SPLINE
SPL {X  -158.454, Y  +360.384, Z    +0.000, E1  +340.634, E3 -446476.060}
SPL {X  -159.737, Y  +373.507, Z    +0.000, E1  +349.689, E3 -446498.095}
SPL {X  -159.990, Y  +382.574, Z    +0.000, E1  +355.537, E3 -446504.783}
SPL {X  -159.990, Y  +389.909, Z    +0.000, E1  +360.662, E3 -446508.797}
SPL {X  -159.990, Y  +396.289, Z    +0.000, E1  +365.500, E3 -446512.577}
SPL {X  -159.990, Y  +407.941, Z    +0.000, E1  +374.126, E3 -446523.914}
SPL {X  -159.990, Y  +418.671, Z    +0.000, E1  +379.855, E3 -446543.330}
SPL {X  -159.990, Y  +429.878, Z    +0.000, E1  +383.330, E3 -446573.386}
SPL {X  -159.990, Y  +432.103, Z    +0.000, E1  +383.301, E3 -446584.404}
SPL {X  -159.990, Y  +434.188, Z    +0.000, E1  +383.325, E3 -446594.601}
SPL {X  -159.990, Y  +437.007, Z    +0.000, E1  +383.323, E3 -446608.492}
SPL {X  -159.990, Y  +439.778, Z    +0.000, E1  +383.323, E3 -446622.124}
SPL {X  -159.990, Y  +442.010, Z    +0.000, E1  +383.308, E3 -446633.145}
SPL {X  -159.990, Y  +443.729, Z    +0.000, E1  +383.310, E3 -446641.601}
SPL {X  -159.990, Y  +446.037, Z    +0.000, E1  +383.324, E3 -446652.938}
SPL {X  -159.990, Y  +448.341, Z    +0.000, E1  +383.317, E3 -446664.256}
SPL {X  -159.990, Y  +450.345, Z    +0.000, E1  +383.316, E3 -446674.134}
SPL {X  -159.990, Y  +452.828, Z    +0.000, E1  +383.330, E3 -446686.333}
SPL {X  -159.990, Y  +456.338, Z    +0.000, E1  +383.359, E3 -446703.525}
SPL {X  -159.990, Y  +459.480, Z    +0.000, E1  +383.323, E3 -446719.067}
SPL {X  -159.990, Y  +461.803, Z    +0.000, E1  +383.322, E3 -446730.502}
SPL {X  -159.990, Y  +464.971, Z    +0.000, E1  +383.357, E3 -446746.008}
SPL {X  -159.990, Y  +467.934, Z    +0.000, E1  +383.321, E3 -446760.665}
SPL {X  -159.990, Y  +469.939, Z    +0.000, E1  +383.319, E3 -446770.527}
SPL {X  -159.990, Y  +472.144, Z    +0.000, E1  +383.327, E3 -446781.378}
SPL {X  -159.990, Y  +474.152, Z    +0.000, E1  +383.309, E3 -446791.330}
SPL {X  -159.990, Y  +476.560, Z    +0.000, E1  +383.332, E3 -446803.138}
SPL {X  -159.990, Y  +478.770, Z    +0.000, E1  +383.306, E3 -446814.063}
SPL {X  -159.990, Y  +480.905, Z    +0.000, E1  +383.327, E3 -446824.531}
SPL {X  -159.990, Y  +484.251, Z    +0.000, E1  +383.352, E3 -446840.947}
SPL {X  -159.990, Y  +488.031, Z    +0.000, E1  +383.345, E3 -446859.579}
SPL {X  -159.990, Y  +491.121, Z    +0.000, E1  +383.323, E3 -446874.825}
SPL {X  -159.990, Y  +493.610, Z    +0.000, E1  +383.323, E3 -446887.078}
SPL {X  -159.990, Y  +496.863, Z    +0.000, E1  +383.350, E3 -446903.038}
SPL {X  -159.990, Y  +499.995, Z    +0.000, E1  +383.324, E3 -446918.499}
SPL {X  -159.990, Y  +502.341, Z    +0.000, E1  +383.320, E3 -446930.058}
SPL {X  -159.990, Y  +505.377, Z    +0.000, E1  +383.346, E3 -446944.949}
SPL {X  -159.990, Y  +508.024, Z    +0.000, E1  +383.315, E3 -446958.031}
SPL {X  -159.990, Y  +510.344, Z    +0.000, E1  +383.327, E3 -446969.438}
SPL {X  -159.990, Y  +513.289, Z    +0.000, E1  +383.332, E3 -446983.928}
SPL {X  -159.990, Y  +516.195, Z    +0.000, E1  +383.325, E3 -446998.247}
SPL {X  -159.990, Y  +518.925, Z    +0.000, E1  +383.333, E3 -447011.610}
SPL {X  -159.990, Y  +521.408, Z    +0.000, E1  +383.329, E3 -447023.819}
SPL {X  -159.990, Y  +523.942, Z    +0.000, E1  +383.333, E3 -447036.312}
SPL {X  -159.990, Y  +527.007, Z    +0.000, E1  +383.339, E3 -447051.412}
SPL {X  -159.990, Y  +529.993, Z    +0.000, E1  +383.329, E3 -447066.114}
SPL {X  -159.990, Y  +532.441, Z    +0.000, E1  +383.322, E3 -447078.165}
SPL {X  -159.990, Y  +534.618, Z    +0.000, E1  +383.322, E3 -447088.898}
SPL {X  -159.990, Y  +537.024, Z    +0.000, E1  +383.321, E3 -447100.760}
SPL {X  -159.990, Y  +539.129, Z    +0.000, E1  +383.310, E3 -447111.143}
SPL {X  -159.990, Y  +541.183, Z    +0.000, E1  +383.319, E3 -447121.240}
SPL {X  -159.990, Y  +543.647, Z    +0.000, E1  +383.325, E3 -447133.343}
SPL {X  -159.990, Y  +546.832, Z    +0.000, E1  +383.349, E3 -447148.966}
SPL {X  -159.990, Y  +549.756, Z    +0.000, E1  +383.320, E3 -447163.407}
SPL {X  -159.990, Y  +551.655, Z    +0.000, E1  +383.320, E3 -447172.758}
SPL {X  -159.990, Y  +553.711, Z    +0.000, E1  +383.317, E3 -447182.879}
SPL {X  -159.990, Y  +555.637, Z    +0.000, E1  +383.323, E3 -447192.348}
SPL {X  -159.990, Y  +558.758, Z    +0.000, E1  +383.351, E3 -447207.658}
SPL {X  -159.990, Y  +561.830, Z    +0.000, E1  +383.325, E3 -447222.831}
SPL {X  -159.990, Y  +564.273, Z    +0.000, E1  +383.325, E3 -447234.855}
SPL {X  -159.990, Y  +567.351, Z    +0.000, E1  +383.348, E3 -447249.951}
SPL {X  -159.990, Y  +570.314, Z    +0.000, E1  +383.326, E3 -447264.583}
SPL {X  -159.990, Y  +572.504, Z    +0.000, E1  +383.321, E3 -447275.368}
SPL {X  -159.990, Y  +575.653, Z    +0.000, E1  +383.355, E3 -447290.805}
SPL {X  -159.990, Y  +578.932, Z    +0.000, E1  +383.330, E3 -447306.988}
SPL {X  -159.990, Y  +581.497, Z    +0.000, E1  +383.329, E3 -447319.572}
SPL {X  -159.990, Y  +583.973, Z    +0.000, E1  +383.332, E3 -447331.757}
SPL {X  -159.990, Y  +586.877, Z    +0.000, E1  +383.349, E3 -447346.012}
SPL {X  -159.990, Y  +590.594, Z    +0.000, E1  +383.363, E3 -447364.262}
SPL {X  -159.990, Y  +593.847, Z    +0.000, E1  +383.340, E3 -447380.273}
SPL {X  -159.990, Y  +596.027, Z    +0.000, E1  +383.330, E3 -447391.019}
SPL {X  -159.990, Y  +599.017, Z    +0.000, E1  +383.373, E3 -447405.584}
SPL {X  -159.990, Y  +601.949, Z    +0.000, E1  +383.344, E3 -447420.035}
SPL {X  -159.990, Y  +604.315, Z    +0.000, E1  +383.350, E3 -447431.661}
SPL {X  -159.990, Y  +607.388, Z    +0.000, E1  +383.369, E3 -447446.725}
SPL {X  -159.990, Y  +610.073, Z    +0.000, E1  +383.343, E3 -447459.991}
SPL {X  -159.990, Y  +612.330, Z    +0.000, E1  +383.340, E3 -447471.118}
SPL {X  -159.990, Y  +615.036, Z    +0.000, E1  +383.353, E3 -447484.405}
SPL {X  -159.990, Y  +618.481, Z    +0.000, E1  +383.366, E3 -447501.343}
SPL {X  -159.990, Y  +621.517, Z    +0.000, E1  +383.337, E3 -447516.326}
SPL {X  -159.990, Y  +623.764, Z    +0.000, E1  +383.335, E3 -447527.377}
SPL {X  -159.990, Y  +626.608, Z    +0.000, E1  +383.361, E3 -447541.302}
SPL {X  -159.990, Y  +630.271, Z    +0.000, E1  +383.375, E3 -447559.263}
SPL {X  -159.990, Y  +633.318, Z    +0.000, E1  +383.339, E3 -447574.340}
SPL {X  -159.990, Y  +635.650, Z    +0.000, E1  +383.339, E3 -447585.811}
SPL {X  -159.990, Y  +638.406, Z    +0.000, E1  +383.354, E3 -447599.378}
SPL {X  -159.990, Y  +641.831, Z    +0.000, E1  +383.342, E3 -447616.325}
SPL {X  -159.990, Y  +644.884, Z    +0.000, E1  +383.324, E3 -447631.412}
SPL {X  -159.990, Y  +647.550, Z    +0.000, E1  +383.318, E3 -447644.579}
SPL {X  -159.990, Y  +650.790, Z    +0.000, E1  +383.346, E3 -447660.446}
SPL {X  -159.990, Y  +654.543, Z    +0.000, E1  +383.348, E3 -447678.899}
SPL {X  -159.990, Y  +658.319, Z    +0.000, E1  +383.349, E3 -447697.488}
SPL {X  -159.990, Y  +661.392, Z    +0.000, E1  +383.318, E3 -447712.691}
SPL {X  -159.990, Y  +663.662, Z    +0.000, E1  +383.322, E3 -447723.815}
SPL {X  -159.990, Y  +665.964, Z    +0.000, E1  +383.328, E3 -447735.106}
SPL {X  -159.990, Y  +667.870, Z    +0.000, E1  +383.320, E3 -447744.513}
SPL {X  -159.990, Y  +669.861, Z    +0.000, E1  +383.321, E3 -447754.314}
SPL {X  -159.990, Y  +671.893, Z    +0.000, E1  +383.319, E3 -447764.322}
SPL {X  -159.974, Y  +673.789, Z    +0.000, E1  +383.323, E3 -447773.638}
SPL {X  -159.924, Y  +676.110, Z    +0.000, E1  +383.320, E3 -447785.122}
SPL {X  -159.801, Y  +679.265, Z    +0.000, E1  +383.327, E3 -447800.741}
SPL {X  -159.626, Y  +682.287, Z    +0.000, E1  +383.280, E3 -447815.839}
SPL {X  -159.462, Y  +684.486, Z    +0.000, E1  +383.258, E3 -447826.839}
SPL {X  -159.289, Y  +686.457, Z    +0.000, E1  +383.223, E3 -447836.749}
SPL {X  -159.052, Y  +688.801, Z    +0.000, E1  +383.217, E3 -447848.484}
SPL {X  -158.658, Y  +692.098, Z    +0.000, E1  +383.176, E3 -447865.109}
ENDSPLINE

SPLINE
SPL {X  -159.063, Y  +688.696, Z    +0.000, E1  +377.094, E3 -447907.328}
SPL {X  -159.957, Y  +674.769, Z    +0.000, E1  +367.092, E3 -447929.709}
SPL {X  -159.990, Y  +671.516, Z    +0.000, E1  +364.944, E3 -447932.095}
SPL {X  -159.990, Y  +663.928, Z    +0.000, E1  +359.662, E3 -447937.187}
SPL {X  -159.990, Y  +658.009, Z    +0.000, E1  +355.226, E3 -447940.887}
SPL {X  -159.990, Y  +651.879, Z    +0.000, E1  +350.548, E3 -447945.949}
SPL {X  -159.990, Y  +637.832, Z    +0.000, E1  +341.694, E3 -447963.540}
SPL {X  -159.990, Y  +626.634, Z    +0.000, E1  +337.968, E3 -447994.394}
SPL {X  -159.990, Y  +624.622, Z    +0.000, E1  +337.980, E3 -448004.977}
SPL {X  -159.990, Y  +622.489, Z    +0.000, E1  +337.969, E3 -448016.144}
SPL {X  -159.990, Y  +619.267, Z    +0.000, E1  +337.938, E3 -448032.978}
SPL {X  -159.990, Y  +615.467, Z    +0.000, E1  +337.940, E3 -448052.914}
SPL {X  -159.990, Y  +612.600, Z    +0.000, E1  +337.975, E3 -448068.025}
SPL {X  -159.990, Y  +610.646, Z    +0.000, E1  +337.979, E3 -448078.282}
SPL {X  -159.990, Y  +608.810, Z    +0.000, E1  +337.977, E3 -448087.915}
SPL {X  -159.990, Y  +606.481, Z    +0.000, E1  +337.967, E3 -448100.091}
SPL {X  -159.990, Y  +603.419, Z    +0.000, E1  +337.936, E3 -448116.030}
SPL {X  -159.990, Y  +600.642, Z    +0.000, E1  +337.968, E3 -448130.660}
SPL {X  -159.990, Y  +598.568, Z    +0.000, E1  +337.954, E3 -448141.452}
SPL {X  -159.990, Y  +595.493, Z    +0.000, E1  +337.930, E3 -448157.536}
SPL {X  -159.990, Y  +592.865, Z    +0.000, E1  +337.964, E3 -448171.364}
SPL {X  -159.990, Y  +590.803, Z    +0.000, E1  +337.954, E3 -448182.155}
SPL {X  -159.990, Y  +588.288, Z    +0.000, E1  +337.950, E3 -448195.319}
SPL {X  -159.990, Y  +586.040, Z    +0.000, E1  +337.954, E3 -448207.064}
SPL {X  -159.990, Y  +584.080, Z    +0.000, E1  +337.953, E3 -448217.324}
SPL {X  -159.990, Y  +581.924, Z    +0.000, E1  +337.949, E3 -448228.624}
SPL {X  -159.990, Y  +579.673, Z    +0.000, E1  +337.950, E3 -448240.423}
SPL {X  -159.990, Y  +576.961, Z    +0.000, E1  +337.936, E3 -448254.602}
SPL {X  -159.990, Y  +574.188, Z    +0.000, E1  +337.947, E3 -448269.149}
SPL {X  -159.990, Y  +571.954, Z    +0.000, E1  +337.959, E3 -448280.907}
SPL {X  -159.990, Y  +570.110, Z    +0.000, E1  +337.958, E3 -448290.557}
SPL {X  -159.990, Y  +568.165, Z    +0.000, E1  +337.957, E3 -448300.737}
SPL {X  -159.990, Y  +565.292, Z    +0.000, E1  +337.922, E3 -448315.715}
SPL {X  -159.990, Y  +562.598, Z    +0.000, E1  +337.958, E3 -448329.926}
SPL {X  -159.990, Y  +560.652, Z    +0.000, E1  +337.962, E3 -448340.138}
SPL {X  -159.990, Y  +558.143, Z    +0.000, E1  +337.928, E3 -448353.170}
SPL {X  -159.990, Y  +555.329, Z    +0.000, E1  +337.943, E3 -448367.914}
SPL {X  -159.990, Y  +553.115, Z    +0.000, E1  +337.946, E3 -448379.520}
SPL {X  -159.990, Y  +550.886, Z    +0.000, E1  +337.944, E3 -448391.201}
SPL {X  -159.990, Y  +548.568, Z    +0.000, E1  +337.944, E3 -448403.322}
SPL {X  -159.990, Y  +545.859, Z    +0.000, E1  +337.926, E3 -448417.472}
SPL {X  -159.990, Y  +542.390, Z    +0.000, E1  +337.914, E3 -448435.642}
SPL {X  -159.990, Y  +539.341, Z    +0.000, E1  +337.944, E3 -448451.664}
SPL {X  -159.990, Y  +536.935, Z    +0.000, E1  +337.942, E3 -448464.253}
SPL {X  -159.990, Y  +534.656, Z    +0.000, E1  +337.946, E3 -448476.197}
SPL {X  -159.990, Y  +531.679, Z    +0.000, E1  +337.913, E3 -448491.711}
SPL {X  -159.990, Y  +527.941, Z    +0.000, E1  +337.907, E3 -448511.253}
SPL {X  -159.990, Y  +525.053, Z    +0.000, E1  +337.942, E3 -448526.443}
SPL {X  -159.990, Y  +522.838, Z    +0.000, E1  +337.933, E3 -448538.048}
SPL {X  -159.990, Y  +519.698, Z    +0.000, E1  +337.916, E3 -448554.431}
SPL {X  -159.990, Y  +517.251, Z    +0.000, E1  +337.946, E3 -448567.291}
SPL {X  -159.990, Y  +515.568, Z    +0.000, E1  +338.084, E3 -448577.388}
ENDSPLINE

SPLINE
SPL {X  -159.990, Y  +517.293, Z    +0.000, E1  +340.923, E3 -448593.686}
ENDSPLINE

SPLINE
SPL {X  -159.990, Y  +512.548, Z    +0.000, E1  +339.587, E3 -448609.261}
SPL {X  -159.990, Y  +508.660, Z    +0.000, E1  +338.515, E3 -448621.315}
SPL {X  -159.990, Y  +503.499, Z    +0.000, E1  +337.116, E3 -448636.395}
SPL {X  -159.990, Y  +498.406, Z    +0.000, E1  +335.789, E3 -448650.427}
SPL {X  -159.990, Y  +494.693, Z    +0.000, E1  +334.929, E3 -448660.895}
SPL {X  -159.990, Y  +491.649, Z    +0.000, E1  +334.596, E3 -448672.097}
SPL {X  -159.990, Y  +488.807, Z    +0.000, E1  +334.603, E3 -448684.822}
SPL {X  -159.990, Y  +486.070, Z    +0.000, E1  +334.601, E3 -448697.053}
SPL {X  -159.990, Y  +483.747, Z    +0.000, E1  +334.616, E3 -448707.466}
SPL {X  -159.990, Y  +481.980, Z    +0.000, E1  +334.616, E3 -448715.363}
SPL {X  -159.990, Y  +479.252, Z    +0.000, E1  +334.588, E3 -448727.505}
SPL {X  -159.990, Y  +475.940, Z    +0.000, E1  +334.597, E3 -448742.325}
SPL {X  -159.990, Y  +473.026, Z    +0.000, E1  +334.601, E3 -448755.355}
SPL {X  -159.990, Y  +470.047, Z    +0.000, E1  +334.598, E3 -448768.673}
SPL {X  -159.990, Y  +466.213, Z    +0.000, E1  +334.567, E3 -448785.753}
SPL {X  -159.990, Y  +462.520, Z    +0.000, E1  +334.600, E3 -448802.321}
SPL {X  -159.990, Y  +460.081, Z    +0.000, E1  +334.610, E3 -448813.223}
SPL {X  -159.990, Y  +457.497, Z    +0.000, E1  +334.597, E3 -448824.747}
SPL {X  -159.990, Y  +455.126, Z    +0.000, E1  +334.611, E3 -448835.356}
SPL {X  -159.990, Y  +452.123, Z    +0.000, E1  +334.574, E3 -448848.713}
SPL {X  -159.990, Y  +448.503, Z    +0.000, E1  +334.590, E3 -448864.915}
SPL {X  -159.990, Y  +445.882, Z    +0.000, E1  +334.615, E3 -448876.717}
SPL {X  -159.990, Y  +443.345, Z    +0.000, E1  +334.610, E3 -448888.100}
SPL {X  -159.990, Y  +441.077, Z    +0.000, E1  +334.631, E3 -448898.298}
SPL {X  -159.990, Y  +438.608, Z    +0.000, E1  +334.608, E3 -448909.295}
SPL {X  -159.990, Y  +435.579, Z    +0.000, E1  +334.614, E3 -448922.849}
SPL {X  -159.990, Y  +432.613, Z    +0.000, E1  +334.610, E3 -448936.116}
SPL {X  -159.990, Y  +429.079, Z    +0.000, E1  +334.593, E3 -448951.887}
SPL {X  -159.990, Y  +426.149, Z    +0.000, E1  +334.626, E3 -448965.049}
SPL {X  -159.990, Y  +423.417, Z    +0.000, E1  +334.600, E3 -448977.214}
SPL {X  -159.990, Y  +419.467, Z    +0.000, E1  +334.583, E3 -448994.849}
SPL {X  -159.990, Y  +416.355, Z    +0.000, E1  +334.625, E3 -449008.846}
SPL {X  -159.990, Y  +413.684, Z    +0.000, E1  +334.603, E3 -449020.753}
SPL {X  -159.990, Y  +410.645, Z    +0.000, E1  +334.615, E3 -449034.365}
SPL {X  -159.990, Y  +408.351, Z    +0.000, E1  +334.628, E3 -449044.651}
SPL {X  -159.990, Y  +406.574, Z    +0.000, E1  +334.625, E3 -449052.568}
SPL {X  -159.990, Y  +404.255, Z    +0.000, E1  +334.609, E3 -449062.904}
SPL {X  -159.990, Y  +401.103, Z    +0.000, E1  +334.596, E3 -449076.968}
SPL {X  -159.990, Y  +398.389, Z    +0.000, E1  +334.619, E3 -449089.164}
SPL {X  -159.990, Y  +395.411, Z    +0.000, E1  +334.600, E3 -449102.461}
SPL {X  -159.990, Y  +392.473, Z    +0.000, E1  +334.623, E3 -449115.646}
SPL {X  -159.990, Y  +390.187, Z    +0.000, E1  +334.622, E3 -449125.904}
SPL {X  -159.990, Y  +387.503, Z    +0.000, E1  +334.622, E3 -449137.899}
SPL {X  -159.990, Y  +384.711, Z    +0.000, E1  +334.612, E3 -449150.343}
SPL {X  -159.988, Y  +381.794, Z    +0.000, E1  +334.611, E3 -449163.378}
SPL {X  -159.958, Y  +379.279, Z    +0.000, E1  +334.625, E3 -449174.668}
SPL {X  -159.867, Y  +376.223, Z    +0.000, E1  +334.608, E3 -449188.383}
SPL {X  -159.727, Y  +373.325, Z    +0.000, E1  +334.659, E3 -449201.547}
SPL {X  -159.549, Y  +370.634, Z    +0.000, E1  +334.653, E3 -449213.721}
SPL {X  -159.201, Y  +366.633, Z    +0.000, E1  +334.686, E3 -449231.913}
SPL {X  -158.798, Y  +363.007, Z    +0.000, E1  +334.761, E3 -449248.570}
SPL {X  -158.453, Y  +360.380, Z    +0.000, E1  +334.828, E3 -449260.715}
SPL {X  -158.127, Y  +358.155, Z    +0.000, E1  +334.874, E3 -449271.046}
SPL {X  -158.095, Y  +357.947, Z    +0.000, E1  +338.259, E3 -449302.618}
ENDSPLINE

SPLINE
SPL {X  -158.454, Y  +360.384, Z    +0.000, E1  +340.634, E3 -449314.769}
SPL {X  -159.737, Y  +373.507, Z    +0.000, E1  +349.689, E3 -449336.805}
SPL {X  -159.990, Y  +382.574, Z    +0.000, E1  +355.537, E3 -449343.492}
SPL {X  -159.990, Y  +387.496, Z    +0.000, E1  +358.996, E3 -449346.237}
SPL {X  -159.990, Y  +395.121, Z    +0.000, E1  +364.514, E3 -449350.550}
SPL {X  -159.990, Y  +407.941, Z    +0.000, E1  +374.126, E3 -449362.624}
SPL {X  -159.990, Y  +418.671, Z    +0.000, E1  +379.855, E3 -449382.040}
SPL {X  -159.990, Y  +429.878, Z    +0.000, E1  +383.330, E3 -449412.095}
SPL {X  -159.990, Y  +432.766, Z    +0.000, E1  +383.321, E3 -449426.318}
SPL {X  -159.990, Y  +434.794, Z    +0.000, E1  +383.304, E3 -449436.349}
SPL {X  -159.990, Y  +437.007, Z    +0.000, E1  +383.323, E3 -449447.201}
SPL {X  -159.990, Y  +439.778, Z    +0.000, E1  +383.323, E3 -449460.834}
SPL {X  -159.990, Y  +442.010, Z    +0.000, E1  +383.308, E3 -449471.855}
SPL {X  -159.990, Y  +443.729, Z    +0.000, E1  +383.310, E3 -449480.311}
SPL {X  -159.990, Y  +446.037, Z    +0.000, E1  +383.324, E3 -449491.648}
SPL {X  -159.990, Y  +448.341, Z    +0.000, E1  +383.317, E3 -449502.966}
SPL {X  -159.990, Y  +450.345, Z    +0.000, E1  +383.316, E3 -449512.844}
SPL {X  -159.990, Y  +452.828, Z    +0.000, E1  +383.330, E3 -449525.043}
SPL {X  -159.990, Y  +456.338, Z    +0.000, E1  +383.359, E3 -449542.235}
SPL {X  -159.990, Y  +459.480, Z    +0.000, E1  +383.323, E3 -449557.777}
SPL {X  -159.990, Y  +461.803, Z    +0.000, E1  +383.322, E3 -449569.212}
SPL {X  -159.990, Y  +464.971, Z    +0.000, E1  +383.357, E3 -449584.718}
SPL {X  -159.990, Y  +467.934, Z    +0.000, E1  +383.321, E3 -449599.375}
SPL {X  -159.990, Y  +469.939, Z    +0.000, E1  +383.319, E3 -449609.237}
SPL {X  -159.990, Y  +472.144, Z    +0.000, E1  +383.327, E3 -449620.087}
SPL {X  -159.990, Y  +474.152, Z    +0.000, E1  +383.309, E3 -449630.039}
SPL {X  -159.990, Y  +476.560, Z    +0.000, E1  +383.332, E3 -449641.847}
SPL {X  -159.990, Y  +478.770, Z    +0.000, E1  +383.306, E3 -449652.773}
SPL {X  -159.990, Y  +480.905, Z    +0.000, E1  +383.327, E3 -449663.241}
SPL {X  -159.990, Y  +484.251, Z    +0.000, E1  +383.352, E3 -449679.656}
SPL {X  -159.990, Y  +488.031, Z    +0.000, E1  +383.345, E3 -449698.289}
SPL {X  -159.990, Y  +491.121, Z    +0.000, E1  +383.323, E3 -449713.535}
SPL {X  -159.990, Y  +493.610, Z    +0.000, E1  +383.323, E3 -449725.788}
SPL {X  -159.990, Y  +496.863, Z    +0.000, E1  +383.350, E3 -449741.748}
SPL {X  -159.990, Y  +499.995, Z    +0.000, E1  +383.324, E3 -449757.209}
SPL {X  -159.990, Y  +502.341, Z    +0.000, E1  +383.320, E3 -449768.768}
SPL {X  -159.990, Y  +504.419, Z    +0.000, E1  +383.313, E3 -449779.010}
SPL {X  -159.990, Y  +507.187, Z    +0.000, E1  +383.346, E3 -449792.563}
SPL {X  -159.990, Y  +510.344, Z    +0.000, E1  +383.327, E3 -449808.148}
SPL {X  -159.990, Y  +512.484, Z    +0.000, E1  +383.309, E3 -449818.720}
SPL {X  -159.990, Y  +514.016, Z    +0.000, E1  +383.308, E3 -449826.269}
SPL {X  -159.990, Y  +516.195, Z    +0.000, E1  +383.325, E3 -449836.957}
SPL {X  -159.990, Y  +518.925, Z    +0.000, E1  +383.333, E3 -449850.320}
SPL {X  -159.990, Y  +521.408, Z    +0.000, E1  +383.329, E3 -449862.529}
SPL {X  -159.990, Y  +523.942, Z    +0.000, E1  +383.333, E3 -449875.022}
SPL {X  -159.990, Y  +527.007, Z    +0.000, E1  +383.339, E3 -449890.121}
SPL {X  -159.990, Y  +529.993, Z    +0.000, E1  +383.329, E3 -449904.824}
SPL {X  -159.990, Y  +532.441, Z    +0.000, E1  +383.322, E3 -449916.874}
SPL {X  -159.990, Y  +534.618, Z    +0.000, E1  +383.322, E3 -449927.608}
SPL {X  -159.990, Y  +537.024, Z    +0.000, E1  +383.321, E3 -449939.470}
SPL {X  -159.990, Y  +539.129, Z    +0.000, E1  +383.310, E3 -449949.853}
SPL {X  -159.990, Y  +541.183, Z    +0.000, E1  +383.319, E3 -449959.950}
SPL {X  -159.990, Y  +543.647, Z    +0.000, E1  +383.325, E3 -449972.053}
SPL {X  -159.990, Y  +546.832, Z    +0.000, E1  +383.349, E3 -449987.675}
SPL {X  -159.990, Y  +549.756, Z    +0.000, E1  +383.320, E3 -450002.116}
SPL {X  -159.990, Y  +551.655, Z    +0.000, E1  +383.320, E3 -450011.467}
SPL {X  -159.990, Y  +553.711, Z    +0.000, E1  +383.317, E3 -450021.589}
SPL {X  -159.990, Y  +556.481, Z    +0.000, E1  +383.354, E3 -450035.151}
SPL {X  -159.990, Y  +559.475, Z    +0.000, E1  +383.321, E3 -450049.956}
SPL {X  -159.990, Y  +561.830, Z    +0.000, E1  +383.325, E3 -450061.541}
SPL {X  -159.990, Y  +564.273, Z    +0.000, E1  +383.325, E3 -450073.565}
SPL {X  -159.990, Y  +566.342, Z    +0.000, E1  +383.314, E3 -450083.770}
SPL {X  -159.990, Y  +568.184, Z    +0.000, E1  +383.317, E3 -450092.830}
SPL {X  -159.990, Y  +570.314, Z    +0.000, E1  +383.326, E3 -450103.293}
SPL {X  -159.990, Y  +573.444, Z    +0.000, E1  +383.356, E3 -450118.632}
SPL {X  -159.990, Y  +577.161, Z    +0.000, E1  +383.346, E3 -450136.956}
SPL {X  -159.990, Y  +580.840, Z    +0.000, E1  +383.355, E3 -450155.006}
SPL {X  -159.990, Y  +583.973, Z    +0.000, E1  +383.332, E3 -450170.467}
SPL {X  -159.990, Y  +586.020, Z    +0.000, E1  +383.323, E3 -450180.551}
SPL {X  -159.990, Y  +587.711, Z    +0.000, E1  +383.318, E3 -450188.891}
SPL {X  -159.990, Y  +589.763, Z    +0.000, E1  +383.328, E3 -450198.967}
SPL {X  -159.990, Y  +591.698, Z    +0.000, E1  +383.324, E3 -450208.452}
SPL {X  -159.990, Y  +593.847, Z    +0.000, E1  +383.340, E3 -450218.982}
SPL {X  -159.990, Y  +597.018, Z    +0.000, E1  +383.367, E3 -450234.514}
SPL {X  -159.990, Y  +599.887, Z    +0.000, E1  +383.341, E3 -450248.619}
SPL {X  -159.990, Y  +601.949, Z    +0.000, E1  +383.344, E3 -450258.745}
SPL {X  -159.990, Y  +605.106, Z    +0.000, E1  +383.383, E3 -450274.191}
SPL {X  -159.990, Y  +608.111, Z    +0.000, E1  +383.342, E3 -450289.042}
SPL {X  -159.990, Y  +610.073, Z    +0.000, E1  +383.343, E3 -450298.700}
SPL {X  -159.990, Y  +612.330, Z    +0.000, E1  +383.340, E3 -450309.828}
SPL {X  -159.990, Y  +615.036, Z    +0.000, E1  +383.353, E3 -450323.115}
SPL {X  -159.990, Y  +618.481, Z    +0.000, E1  +383.366, E3 -450340.053}
SPL {X  -159.990, Y  +621.517, Z    +0.000, E1  +383.337, E3 -450355.036}
SPL {X  -159.990, Y  +623.764, Z    +0.000, E1  +383.335, E3 -450366.086}
SPL {X  -159.990, Y  +626.608, Z    +0.000, E1  +383.361, E3 -450380.011}
SPL {X  -159.990, Y  +630.271, Z    +0.000, E1  +383.375, E3 -450397.973}
SPL {X  -159.990, Y  +633.318, Z    +0.000, E1  +383.339, E3 -450413.050}
SPL {X  -159.990, Y  +635.650, Z    +0.000, E1  +383.339, E3 -450424.521}
SPL {X  -159.990, Y  +638.406, Z    +0.000, E1  +383.354, E3 -450438.088}
SPL {X  -159.990, Y  +641.831, Z    +0.000, E1  +383.342, E3 -450455.035}
SPL {X  -159.990, Y  +644.884, Z    +0.000, E1  +383.324, E3 -450470.122}
SPL {X  -159.990, Y  +647.550, Z    +0.000, E1  +383.318, E3 -450483.289}
SPL {X  -159.990, Y  +650.790, Z    +0.000, E1  +383.346, E3 -450499.155}
SPL {X  -159.990, Y  +654.543, Z    +0.000, E1  +383.348, E3 -450517.608}
SPL {X  -159.990, Y  +658.319, Z    +0.000, E1  +383.349, E3 -450536.198}
SPL {X  -159.990, Y  +661.392, Z    +0.000, E1  +383.318, E3 -450551.401}
SPL {X  -159.990, Y  +663.662, Z    +0.000, E1  +383.322, E3 -450562.525}
SPL {X  -159.990, Y  +665.964, Z    +0.000, E1  +383.328, E3 -450573.815}
SPL {X  -159.990, Y  +667.870, Z    +0.000, E1  +383.320, E3 -450583.222}
SPL {X  -159.990, Y  +669.861, Z    +0.000, E1  +383.321, E3 -450593.023}
SPL {X  -159.983, Y  +672.946, Z    +0.000, E1  +383.359, E3 -450608.133}
SPL {X  -159.924, Y  +676.110, Z    +0.000, E1  +383.320, E3 -450623.832}
SPL {X  -159.845, Y  +678.302, Z    +0.000, E1  +383.298, E3 -450634.734}
SPL {X  -159.760, Y  +680.081, Z    +0.000, E1  +383.288, E3 -450643.577}
SPL {X  -159.626, Y  +682.287, Z    +0.000, E1  +383.280, E3 -450654.549}
SPL {X  -159.462, Y  +684.486, Z    +0.000, E1  +383.258, E3 -450665.548}
SPL {X  -159.212, Y  +687.262, Z    +0.000, E1  +383.238, E3 -450679.452}
SPL {X  -158.971, Y  +689.529, Z    +0.000, E1  +383.181, E3 -450690.912}
SPL {X  -158.658, Y  +692.098, Z    +0.000, E1  +383.176, E3 -450703.819}
ENDSPLINE

SPLINE
SPL {X  -159.063, Y  +688.696, Z    +0.000, E1  +377.094, E3 -450746.037}
SPL {X  -159.987, Y  +672.488, Z    +0.000, E1  +365.638, E3 -450770.102}
SPL {X  -159.990, Y  +663.928, Z    +0.000, E1  +359.662, E3 -450775.897}
SPL {X  -159.990, Y  +658.009, Z    +0.000, E1  +355.226, E3 -450779.597}
SPL {X  -159.990, Y  +651.879, Z    +0.000, E1  +350.548, E3 -450784.659}
SPL {X  -159.990, Y  +637.832, Z    +0.000, E1  +341.694, E3 -450802.250}
SPL {X  -159.990, Y  +626.634, Z    +0.000, E1  +337.968, E3 -450833.103}
SPL {X  -159.990, Y  +624.622, Z    +0.000, E1  +337.980, E3 -450843.687}
SPL {X  -159.990, Y  +622.489, Z    +0.000, E1  +337.969, E3 -450854.853}
SPL {X  -159.990, Y  +619.955, Z    +0.000, E1  +337.968, E3 -450868.143}
SPL {X  -159.990, Y  +617.386, Z    +0.000, E1  +337.968, E3 -450881.618}
SPL {X  -159.990, Y  +614.863, Z    +0.000, E1  +337.969, E3 -450894.850}
SPL {X  -159.990, Y  +612.600, Z    +0.000, E1  +337.975, E3 -450906.734}
SPL {X  -159.990, Y  +610.646, Z    +0.000, E1  +337.979, E3 -450916.992}
SPL {X  -159.990, Y  +608.810, Z    +0.000, E1  +337.977, E3 -450926.625}
SPL {X  -159.990, Y  +605.804, Z    +0.000, E1  +337.936, E3 -450942.270}
SPL {X  -159.990, Y  +602.819, Z    +0.000, E1  +337.963, E3 -450957.941}
SPL {X  -159.990, Y  +600.642, Z    +0.000, E1  +337.968, E3 -450969.369}
SPL {X  -159.990, Y  +598.568, Z    +0.000, E1  +337.954, E3 -450980.162}
SPL {X  -159.990, Y  +596.440, Z    +0.000, E1  +337.964, E3 -450991.344}
SPL {X  -159.990, Y  +593.768, Z    +0.000, E1  +337.929, E3 -451005.276}
SPL {X  -159.990, Y  +590.068, Z    +0.000, E1  +337.924, E3 -451024.645}
SPL {X  -159.990, Y  +586.620, Z    +0.000, E1  +337.935, E3 -451042.707}
SPL {X  -159.990, Y  +584.080, Z    +0.000, E1  +337.953, E3 -451056.034}
SPL {X  -159.990, Y  +581.924, Z    +0.000, E1  +337.949, E3 -451067.334}
SPL {X  -159.990, Y  +578.886, Z    +0.000, E1  +337.918, E3 -451083.188}
SPL {X  -159.990, Y  +576.252, Z    +0.000, E1  +337.962, E3 -451097.086}
SPL {X  -159.990, Y  +574.188, Z    +0.000, E1  +337.947, E3 -451107.859}
SPL {X  -159.990, Y  +571.954, Z    +0.000, E1  +337.959, E3 -451119.617}
SPL {X  -159.990, Y  +570.110, Z    +0.000, E1  +337.958, E3 -451129.267}
SPL {X  -159.990, Y  +568.165, Z    +0.000, E1  +337.957, E3 -451139.447}
SPL {X  -159.990, Y  +566.106, Z    +0.000, E1  +337.954, E3 -451150.230}
SPL {X  -159.990, Y  +563.259, Z    +0.000, E1  +337.929, E3 -451165.112}
SPL {X  -159.990, Y  +559.661, Z    +0.000, E1  +337.922, E3 -451183.935}
SPL {X  -159.990, Y  +555.965, Z    +0.000, E1  +337.915, E3 -451203.244}
SPL {X  -159.990, Y  +553.115, Z    +0.000, E1  +337.946, E3 -451218.229}
SPL {X  -159.990, Y  +550.886, Z    +0.000, E1  +337.944, E3 -451229.911}
SPL {X  -159.990, Y  +548.568, Z    +0.000, E1  +337.944, E3 -451242.032}
SPL {X  -159.990, Y  +545.859, Z    +0.000, E1  +337.926, E3 -451256.181}
SPL {X  -159.990, Y  +543.060, Z    +0.000, E1  +337.943, E3 -451270.905}
SPL {X  -159.990, Y  +539.928, Z    +0.000, E1  +337.917, E3 -451287.246}
SPL {X  -159.990, Y  +536.935, Z    +0.000, E1  +337.942, E3 -451302.963}
SPL {X  -159.990, Y  +534.656, Z    +0.000, E1  +337.946, E3 -451314.907}
SPL {X  -159.990, Y  +531.679, Z    +0.000, E1  +337.913, E3 -451330.421}
SPL {X  -159.990, Y  +527.941, Z    +0.000, E1  +337.907, E3 -451349.963}
SPL {X  -159.990, Y  +525.053, Z    +0.000, E1  +337.942, E3 -451365.153}
SPL {X  -159.990, Y  +522.838, Z    +0.000, E1  +337.933, E3 -451376.757}
SPL {X  -159.990, Y  +519.698, Z    +0.000, E1  +337.916, E3 -451393.140}
SPL {X  -159.990, Y  +517.251, Z    +0.000, E1  +337.946, E3 -451406.000}
SPL {X  -159.990, Y  +515.568, Z    +0.000, E1  +338.084, E3 -451416.097}
ENDSPLINE

SPLINE
SPL {X  -159.990, Y  +517.293, Z    +0.000, E1  +340.923, E3 -451432.396}
ENDSPLINE

SPLINE
SPL {X  -159.990, Y  +512.548, Z    +0.000, E1  +339.587, E3 -451447.971}
SPL {X  -159.990, Y  +508.660, Z    +0.000, E1  +338.515, E3 -451460.025}
SPL {X  -159.990, Y  +503.499, Z    +0.000, E1  +337.116, E3 -451475.104}
SPL {X  -159.990, Y  +498.406, Z    +0.000, E1  +335.789, E3 -451489.137}
SPL {X  -159.990, Y  +494.693, Z    +0.000, E1  +334.929, E3 -451499.604}
SPL {X  -159.990, Y  +491.649, Z    +0.000, E1  +334.596, E3 -451510.807}
SPL {X  -159.990, Y  +488.807, Z    +0.000, E1  +334.603, E3 -451523.531}
SPL {X  -159.990, Y  +486.070, Z    +0.000, E1  +334.601, E3 -451535.762}
SPL {X  -159.990, Y  +482.821, Z    +0.000, E1  +334.589, E3 -451550.264}
SPL {X  -159.990, Y  +480.183, Z    +0.000, E1  +334.616, E3 -451562.104}
SPL {X  -159.990, Y  +478.407, Z    +0.000, E1  +334.616, E3 -451570.044}
SPL {X  -159.990, Y  +475.940, Z    +0.000, E1  +334.597, E3 -451581.035}
SPL {X  -159.990, Y  +473.026, Z    +0.000, E1  +334.601, E3 -451594.064}
SPL {X  -159.990, Y  +470.047, Z    +0.000, E1  +334.598, E3 -451607.383}
SPL {X  -159.990, Y  +467.082, Z    +0.000, E1  +334.601, E3 -451620.630}
SPL {X  -159.990, Y  +464.919, Z    +0.000, E1  +334.619, E3 -451630.357}
SPL {X  -159.990, Y  +462.520, Z    +0.000, E1  +334.600, E3 -451641.031}
SPL {X  -159.990, Y  +460.081, Z    +0.000, E1  +334.610, E3 -451651.933}
SPL {X  -159.990, Y  +457.497, Z    +0.000, E1  +334.597, E3 -451663.457}
SPL {X  -159.990, Y  +454.323, Z    +0.000, E1  +334.588, E3 -451677.616}
SPL {X  -159.990, Y  +451.400, Z    +0.000, E1  +334.603, E3 -451690.707}
SPL {X  -159.990, Y  +448.503, Z    +0.000, E1  +334.590, E3 -451703.625}
SPL {X  -159.990, Y  +445.108, Z    +0.000, E1  +334.593, E3 -451718.863}
SPL {X  -159.990, Y  +441.797, Z    +0.000, E1  +334.610, E3 -451733.742}
SPL {X  -159.990, Y  +439.442, Z    +0.000, E1  +334.631, E3 -451744.319}
SPL {X  -159.990, Y  +436.316, Z    +0.000, E1  +334.580, E3 -451758.201}
SPL {X  -159.990, Y  +432.613, Z    +0.000, E1  +334.610, E3 -451774.826}
SPL {X  -159.990, Y  +429.079, Z    +0.000, E1  +334.593, E3 -451790.597}
SPL {X  -159.990, Y  +426.149, Z    +0.000, E1  +334.626, E3 -451803.759}
SPL {X  -159.990, Y  +423.417, Z    +0.000, E1  +334.600, E3 -451815.924}
SPL {X  -159.990, Y  +419.467, Z    +0.000, E1  +334.583, E3 -451833.559}
SPL {X  -159.990, Y  +416.355, Z    +0.000, E1  +334.625, E3 -451847.556}
SPL {X  -159.990, Y  +413.684, Z    +0.000, E1  +334.603, E3 -451859.463}
SPL {X  -159.990, Y  +410.645, Z    +0.000, E1  +334.615, E3 -451873.075}
SPL {X  -159.990, Y  +408.351, Z    +0.000, E1  +334.628, E3 -451883.361}
SPL {X  -159.990, Y  +406.574, Z    +0.000, E1  +334.625, E3 -451891.277}
SPL {X  -159.990, Y  +404.255, Z    +0.000, E1  +334.609, E3 -451901.614}
SPL {X  -159.990, Y  +401.103, Z    +0.000, E1  +334.596, E3 -451915.678}
SPL {X  -159.990, Y  +398.389, Z    +0.000, E1  +334.619, E3 -451927.874}
SPL {X  -159.990, Y  +395.411, Z    +0.000, E1  +334.600, E3 -451941.171}
SPL {X  -159.990, Y  +392.473, Z    +0.000, E1  +334.623, E3 -451954.356}
SPL {X  -159.990, Y  +390.187, Z    +0.000, E1  +334.622, E3 -451964.614}
SPL {X  -159.990, Y  +387.503, Z    +0.000, E1  +334.622, E3 -451976.609}
SPL {X  -159.990, Y  +384.711, Z    +0.000, E1  +334.612, E3 -451989.053}
SPL {X  -159.988, Y  +381.794, Z    +0.000, E1  +334.611, E3 -452002.088}
SPL {X  -159.958, Y  +379.279, Z    +0.000, E1  +334.625, E3 -452013.378}
SPL {X  -159.894, Y  +376.959, Z    +0.000, E1  +334.630, E3 -452023.822}
SPL {X  -159.765, Y  +374.027, Z    +0.000, E1  +334.633, E3 -452037.038}
SPL {X  -159.607, Y  +371.442, Z    +0.000, E1  +334.673, E3 -452048.813}
SPL {X  -159.379, Y  +368.534, Z    +0.000, E1  +334.684, E3 -452062.000}
SPL {X  -159.113, Y  +365.767, Z    +0.000, E1  +334.734, E3 -452074.640}
SPL {X  -158.869, Y  +363.595, Z    +0.000, E1  +334.770, E3 -452084.611}
SPL {X  -158.527, Y  +360.915, Z    +0.000, E1  +334.798, E3 -452096.917}
SPL {X  -158.127, Y  +358.155, Z    +0.000, E1  +334.874, E3 -452109.755}
SPL {X  -158.095, Y  +357.947, Z    +0.000, E1  +338.259, E3 -452141.328}
ENDSPLINE

SPLINE
SPL {X  -158.454, Y  +360.384, Z    +0.000, E1  +340.634, E3 -452153.479}
SPL {X  -159.737, Y  +373.507, Z    +0.000, E1  +349.689, E3 -452175.514}
SPL {X  -159.990, Y  +382.574, Z    +0.000, E1  +355.537, E3 -452182.202}
SPL {X  -159.990, Y  +387.496, Z    +0.000, E1  +358.996, E3 -452184.947}
SPL {X  -159.990, Y  +395.121, Z    +0.000, E1  +364.514, E3 -452189.259}
SPL {X  -159.990, Y  +407.941, Z    +0.000, E1  +374.126, E3 -452201.334}
SPL {X  -159.990, Y  +418.671, Z    +0.000, E1  +379.855, E3 -452220.750}
SPL {X  -159.990, Y  +429.878, Z    +0.000, E1  +383.330, E3 -452250.805}
SPL {X  -159.990, Y  +432.103, Z    +0.000, E1  +383.301, E3 -452261.823}
SPL {X  -159.990, Y  +434.188, Z    +0.000, E1  +383.325, E3 -452272.020}
SPL {X  -159.990, Y  +436.320, Z    +0.000, E1  +383.304, E3 -452282.573}
SPL {X  -159.990, Y  +439.169, Z    +0.000, E1  +383.353, E3 -452296.490}
SPL {X  -159.990, Y  +442.945, Z    +0.000, E1  +383.339, E3 -452315.107}
SPL {X  -159.990, Y  +446.037, Z    +0.000, E1  +383.324, E3 -452330.358}
SPL {X  -159.990, Y  +448.341, Z    +0.000, E1  +383.317, E3 -452341.675}
SPL {X  -159.990, Y  +450.345, Z    +0.000, E1  +383.316, E3 -452351.553}
SPL {X  -159.990, Y  +452.828, Z    +0.000, E1  +383.330, E3 -452363.753}
SPL {X  -159.990, Y  +456.338, Z    +0.000, E1  +383.359, E3 -452380.945}
SPL {X  -159.990, Y  +459.480, Z    +0.000, E1  +383.323, E3 -452396.486}
SPL {X  -159.990, Y  +461.803, Z    +0.000, E1  +383.322, E3 -452407.921}
SPL {X  -159.990, Y  +464.971, Z    +0.000, E1  +383.357, E3 -452423.427}
SPL {X  -159.990, Y  +467.934, Z    +0.000, E1  +383.321, E3 -452438.085}
SPL {X  -159.990, Y  +469.939, Z    +0.000, E1  +383.319, E3 -452447.946}
SPL {X  -159.990, Y  +472.144, Z    +0.000, E1  +383.327, E3 -452458.797}
SPL {X  -159.990, Y  +474.152, Z    +0.000, E1  +383.309, E3 -452468.749}
SPL {X  -159.990, Y  +475.762, Z    +0.000, E1  +383.308, E3 -452476.678}
SPL {X  -159.990, Y  +478.041, Z    +0.000, E1  +383.328, E3 -452487.854}
SPL {X  -159.990, Y  +480.905, Z    +0.000, E1  +383.327, E3 -452501.950}
SPL {X  -159.990, Y  +483.391, Z    +0.000, E1  +383.320, E3 -452514.191}
SPL {X  -159.990, Y  +485.299, Z    +0.000, E1  +383.310, E3 -452523.620}
SPL {X  -159.990, Y  +487.362, Z    +0.000, E1  +383.320, E3 -452533.753}
SPL {X  -159.990, Y  +490.503, Z    +0.000, E1  +383.351, E3 -452549.149}
SPL {X  -159.990, Y  +493.610, Z    +0.000, E1  +383.323, E3 -452564.497}
SPL {X  -159.990, Y  +495.794, Z    +0.000, E1  +383.312, E3 -452575.271}
SPL {X  -159.990, Y  +497.668, Z    +0.000, E1  +383.317, E3 -452584.481}
SPL {X  -159.990, Y  +499.995, Z    +0.000, E1  +383.324, E3 -452595.919}
SPL {X  -159.990, Y  +502.341, Z    +0.000, E1  +383.320, E3 -452607.478}
SPL {X  -159.990, Y  +504.419, Z    +0.000, E1  +383.313, E3 -452617.719}
SPL {X  -159.990, Y  +506.252, Z    +0.000, E1  +383.313, E3 -452626.745}
SPL {X  -159.990, Y  +508.697, Z    +0.000, E1  +383.335, E3 -452638.728}
SPL {X  -159.990, Y  +511.771, Z    +0.000, E1  +383.331, E3 -452653.875}
SPL {X  -159.990, Y  +514.016, Z    +0.000, E1  +383.308, E3 -452664.978}
SPL {X  -159.990, Y  +516.195, Z    +0.000, E1  +383.325, E3 -452675.666}
SPL {X  -159.990, Y  +518.925, Z    +0.000, E1  +383.333, E3 -452689.030}
SPL {X  -159.990, Y  +521.408, Z    +0.000, E1  +383.329, E3 -452701.239}
SPL {X  -159.990, Y  +523.942, Z    +0.000, E1  +383.333, E3 -452713.731}
SPL {X  -159.990, Y  +526.221, Z    +0.000, E1  +383.314, E3 -452725.007}
SPL {X  -159.990, Y  +527.834, Z    +0.000, E1  +383.311, E3 -452732.957}
SPL {X  -159.990, Y  +529.993, Z    +0.000, E1  +383.329, E3 -452743.533}
SPL {X  -159.990, Y  +532.441, Z    +0.000, E1  +383.322, E3 -452755.584}
SPL {X  -159.990, Y  +534.618, Z    +0.000, E1  +383.322, E3 -452766.317}
SPL {X  -159.990, Y  +537.024, Z    +0.000, E1  +383.321, E3 -452778.180}
SPL {X  -159.990, Y  +539.129, Z    +0.000, E1  +383.310, E3 -452788.562}
SPL {X  -159.990, Y  +541.183, Z    +0.000, E1  +383.319, E3 -452798.659}
SPL {X  -159.990, Y  +543.647, Z    +0.000, E1  +383.325, E3 -452810.762}
SPL {X  -159.990, Y  +546.832, Z    +0.000, E1  +383.349, E3 -452826.385}
SPL {X  -159.990, Y  +549.756, Z    +0.000, E1  +383.320, E3 -452840.826}
SPL {X  -159.990, Y  +551.655, Z    +0.000, E1  +383.320, E3 -452850.177}
SPL {X  -159.990, Y  +553.711, Z    +0.000, E1  +383.317, E3 -452860.299}
SPL {X  -159.990, Y  +555.637, Z    +0.000, E1  +383.323, E3 -452869.768}
SPL {X  -159.990, Y  +558.758, Z    +0.000, E1  +383.351, E3 -452885.077}
SPL {X  -159.990, Y  +561.830, Z    +0.000, E1  +383.325, E3 -452900.250}
SPL {X  -159.990, Y  +564.273, Z    +0.000, E1  +383.325, E3 -452912.275}
SPL {X  -159.990, Y  +567.351, Z    +0.000, E1  +383.348, E3 -452927.371}
SPL {X  -159.990, Y  +570.314, Z    +0.000, E1  +383.326, E3 -452942.003}
SPL {X  -159.990, Y  +572.504, Z    +0.000, E1  +383.321, E3 -452952.788}
SPL {X  -159.990, Y  +575.653, Z    +0.000, E1  +383.355, E3 -452968.224}
SPL {X  -159.990, Y  +578.932, Z    +0.000, E1  +383.330, E3 -452984.407}
SPL {X  -159.990, Y  +581.497, Z    +0.000, E1  +383.329, E3 -452996.992}
SPL {X  -159.990, Y  +583.973, Z    +0.000, E1  +383.332, E3 -453009.177}
SPL {X  -159.990, Y  +586.020, Z    +0.000, E1  +383.323, E3 -453019.261}
SPL {X  -159.990, Y  +587.711, Z    +0.000, E1  +383.318, E3 -453027.600}
SPL {X  -159.990, Y  +589.763, Z    +0.000, E1  +383.328, E3 -453037.677}
SPL {X  -159.990, Y  +591.698, Z    +0.000, E1  +383.324, E3 -453047.161}
SPL {X  -159.990, Y  +593.847, Z    +0.000, E1  +383.340, E3 -453057.692}
SPL {X  -159.990, Y  +597.018, Z    +0.000, E1  +383.367, E3 -453073.224}
SPL {X  -159.990, Y  +599.887, Z    +0.000, E1  +383.341, E3 -453087.328}
SPL {X  -159.990, Y  +601.949, Z    +0.000, E1  +383.344, E3 -453097.455}
SPL {X  -159.990, Y  +605.106, Z    +0.000, E1  +383.383, E3 -453112.901}
SPL {X  -159.990, Y  +608.111, Z    +0.000, E1  +383.342, E3 -453127.752}
SPL {X  -159.990, Y  +610.073, Z    +0.000, E1  +383.343, E3 -453137.410}
SPL {X  -159.990, Y  +612.330, Z    +0.000, E1  +383.340, E3 -453148.537}
SPL {X  -159.990, Y  +615.036, Z    +0.000, E1  +383.353, E3 -453161.825}
SPL {X  -159.990, Y  +618.481, Z    +0.000, E1  +383.366, E3 -453178.763}
SPL {X  -159.990, Y  +621.517, Z    +0.000, E1  +383.337, E3 -453193.746}
SPL {X  -159.990, Y  +623.764, Z    +0.000, E1  +383.335, E3 -453204.796}
SPL {X  -159.990, Y  +626.608, Z    +0.000, E1  +383.361, E3 -453218.721}
SPL {X  -159.990, Y  +630.271, Z    +0.000, E1  +383.375, E3 -453236.682}
SPL {X  -159.990, Y  +633.318, Z    +0.000, E1  +383.339, E3 -453251.760}
SPL {X  -159.990, Y  +635.650, Z    +0.000, E1  +383.339, E3 -453263.231}
SPL {X  -159.990, Y  +638.406, Z    +0.000, E1  +383.354, E3 -453276.797}
SPL {X  -159.990, Y  +641.831, Z    +0.000, E1  +383.342, E3 -453293.745}
SPL {X  -159.990, Y  +644.884, Z    +0.000, E1  +383.324, E3 -453308.832}
SPL {X  -159.990, Y  +647.550, Z    +0.000, E1  +383.318, E3 -453321.998}
SPL {X  -159.990, Y  +650.790, Z    +0.000, E1  +383.346, E3 -453337.865}
SPL {X  -159.990, Y  +654.543, Z    +0.000, E1  +383.348, E3 -453356.318}
SPL {X  -159.990, Y  +658.319, Z    +0.000, E1  +383.349, E3 -453374.908}
SPL {X  -159.990, Y  +661.392, Z    +0.000, E1  +383.318, E3 -453390.111}
SPL {X  -159.990, Y  +663.662, Z    +0.000, E1  +383.322, E3 -453401.235}
SPL {X  -159.990, Y  +665.964, Z    +0.000, E1  +383.328, E3 -453412.525}
SPL {X  -159.990, Y  +667.870, Z    +0.000, E1  +383.320, E3 -453421.932}
SPL {X  -159.990, Y  +669.861, Z    +0.000, E1  +383.321, E3 -453431.733}
SPL {X  -159.990, Y  +671.893, Z    +0.000, E1  +383.319, E3 -453441.741}
SPL {X  -159.974, Y  +673.789, Z    +0.000, E1  +383.323, E3 -453451.057}
SPL {X  -159.924, Y  +676.110, Z    +0.000, E1  +383.320, E3 -453462.541}
SPL {X  -159.801, Y  +679.265, Z    +0.000, E1  +383.327, E3 -453478.160}
SPL {X  -159.626, Y  +682.287, Z    +0.000, E1  +383.280, E3 -453493.259}
SPL {X  -159.462, Y  +684.486, Z    +0.000, E1  +383.258, E3 -453504.258}
SPL {X  -159.212, Y  +687.262, Z    +0.000, E1  +383.238, E3 -453518.162}
SPL {X  -158.971, Y  +689.529, Z    +0.000, E1  +383.181, E3 -453529.622}
SPL {X  -158.658, Y  +692.098, Z    +0.000, E1  +383.176, E3 -453542.528}
ENDSPLINE

SPLINE
SPL {X  -159.063, Y  +688.696, Z    +0.000, E1  +377.094, E3 -453584.747}
SPL {X  -159.957, Y  +674.769, Z    +0.000, E1  +367.092, E3 -453607.129}
SPL {X  -159.990, Y  +671.516, Z    +0.000, E1  +364.944, E3 -453609.515}
SPL {X  -159.990, Y  +663.928, Z    +0.000, E1  +359.662, E3 -453614.606}
SPL {X  -159.990, Y  +658.009, Z    +0.000, E1  +355.226, E3 -453618.306}
SPL {X  -159.990, Y  +651.879, Z    +0.000, E1  +350.548, E3 -453623.369}
SPL {X  -159.990, Y  +637.832, Z    +0.000, E1  +341.694, E3 -453640.960}
SPL {X  -159.990, Y  +626.634, Z    +0.000, E1  +337.968, E3 -453671.813}
SPL {X  -159.990, Y  +624.622, Z    +0.000, E1  +337.980, E3 -453682.397}
SPL {X  -159.990, Y  +622.489, Z    +0.000, E1  +337.969, E3 -453693.563}
SPL {X  -159.990, Y  +619.267, Z    +0.000, E1  +337.938, E3 -453710.397}
SPL {X  -159.990, Y  +615.467, Z    +0.000, E1  +337.940, E3 -453730.334}
SPL {X  -159.990, Y  +612.600, Z    +0.000, E1  +337.975, E3 -453745.444}
SPL {X  -159.990, Y  +610.646, Z    +0.000, E1  +337.979, E3 -453755.702}
SPL {X  -159.990, Y  +608.810, Z    +0.000, E1  +337.977, E3 -453765.334}
SPL {X  -159.990, Y  +605.804, Z    +0.000, E1  +337.936, E3 -453780.980}
SPL {X  -159.990, Y  +602.819, Z    +0.000, E1  +337.963, E3 -453796.651}
SPL {X  -159.990, Y  +600.642, Z    +0.000, E1  +337.968, E3 -453808.079}
SPL {X  -159.990, Y  +598.568, Z    +0.000, E1  +337.954, E3 -453818.872}
SPL {X  -159.990, Y  +596.440, Z    +0.000, E1  +337.964, E3 -453830.053}
SPL {X  -159.990, Y  +593.768, Z    +0.000, E1  +337.929, E3 -453843.986}
SPL {X  -159.990, Y  +590.068, Z    +0.000, E1  +337.924, E3 -453863.355}
SPL {X  -159.990, Y  +586.620, Z    +0.000, E1  +337.935, E3 -453881.417}
SPL {X  -159.990, Y  +584.080, Z    +0.000, E1  +337.953, E3 -453894.743}
SPL {X  -159.990, Y  +581.924, Z    +0.000, E1  +337.949, E3 -453906.044}
SPL {X  -159.990, Y  +578.886, Z    +0.000, E1  +337.918, E3 -453921.898}
SPL {X  -159.990, Y  +576.252, Z    +0.000, E1  +337.962, E3 -453935.796}
SPL {X  -159.990, Y  +574.188, Z    +0.000, E1  +337.947, E3 -453946.569}
SPL {X  -159.990, Y  +571.954, Z    +0.000, E1  +337.959, E3 -453958.326}
SPL {X  -159.990, Y  +570.110, Z    +0.000, E1  +337.958, E3 -453967.977}
SPL {X  -159.990, Y  +568.165, Z    +0.000, E1  +337.957, E3 -453978.156}
SPL {X  -159.990, Y  +565.292, Z    +0.000, E1  +337.922, E3 -453993.134}
SPL {X  -159.990, Y  +562.598, Z    +0.000, E1  +337.958, E3 -454007.346}
SPL {X  -159.990, Y  +560.652, Z    +0.000, E1  +337.962, E3 -454017.558}
SPL {X  -159.990, Y  +558.143, Z    +0.000, E1  +337.928, E3 -454030.589}
SPL {X  -159.990, Y  +555.329, Z    +0.000, E1  +337.943, E3 -454045.334}
SPL {X  -159.990, Y  +553.115, Z    +0.000, E1  +337.946, E3 -454056.939}
SPL {X  -159.990, Y  +550.886, Z    +0.000, E1  +337.944, E3 -454068.620}
SPL {X  -159.990, Y  +548.568, Z    +0.000, E1  +337.944, E3 -454080.741}
SPL {X  -159.990, Y  +545.859, Z    +0.000, E1  +337.926, E3 -454094.891}
SPL {X  -159.990, Y  +542.390, Z    +0.000, E1  +337.914, E3 -454113.062}
SPL {X  -159.990, Y  +539.341, Z    +0.000, E1  +337.944, E3 -454129.083}
SPL {X  -159.990, Y  +536.935, Z    +0.000, E1  +337.942, E3 -454141.673}
SPL {X  -159.990, Y  +534.656, Z    +0.000, E1  +337.946, E3 -454153.616}
SPL {X  -159.990, Y  +531.679, Z    +0.000, E1  +337.913, E3 -454169.130}
SPL {X  -159.990, Y  +527.941, Z    +0.000, E1  +337.907, E3 -454188.673}
SPL {X  -159.990, Y  +525.053, Z    +0.000, E1  +337.942, E3 -454203.863}
SPL {X  -159.990, Y  +522.838, Z    +0.000, E1  +337.933, E3 -454215.467}
SPL {X  -159.990, Y  +519.698, Z    +0.000, E1  +337.916, E3 -454231.850}
SPL {X  -159.990, Y  +517.251, Z    +0.000, E1  +337.946, E3 -454244.710}
SPL {X  -159.990, Y  +515.568, Z    +0.000, E1  +338.084, E3 -454254.807}
ENDSPLINE

SPLINE
SPL {X  -159.990, Y  +517.293, Z    +0.000, E1  +340.923, E3 -454271.105}
ENDSPLINE

SPLINE
SPL {X  -159.990, Y  +512.548, Z    +0.000, E1  +339.587, E3 -454286.680}
SPL {X  -159.990, Y  +508.660, Z    +0.000, E1  +338.515, E3 -454298.735}
SPL {X  -159.990, Y  +503.499, Z    +0.000, E1  +337.116, E3 -454313.814}
SPL {X  -159.990, Y  +498.406, Z    +0.000, E1  +335.789, E3 -454327.847}
SPL {X  -159.990, Y  +494.693, Z    +0.000, E1  +334.929, E3 -454338.314}
SPL {X  -159.990, Y  +491.649, Z    +0.000, E1  +334.596, E3 -454349.517}
SPL {X  -159.990, Y  +488.807, Z    +0.000, E1  +334.603, E3 -454362.241}
SPL {X  -159.990, Y  +486.070, Z    +0.000, E1  +334.601, E3 -454374.472}
SPL {X  -159.990, Y  +483.747, Z    +0.000, E1  +334.616, E3 -454384.885}
SPL {X  -159.990, Y  +481.038, Z    +0.000, E1  +334.588, E3 -454396.940}
SPL {X  -159.990, Y  +477.508, Z    +0.000, E1  +334.590, E3 -454412.722}
SPL {X  -159.990, Y  +473.634, Z    +0.000, E1  +334.574, E3 -454430.012}
SPL {X  -159.990, Y  +470.047, Z    +0.000, E1  +334.598, E3 -454446.093}
SPL {X  -159.990, Y  +467.082, Z    +0.000, E1  +334.601, E3 -454459.340}
SPL {X  -159.990, Y  +464.063, Z    +0.000, E1  +334.595, E3 -454472.835}
SPL {X  -159.990, Y  +460.712, Z    +0.000, E1  +334.589, E3 -454487.794}
SPL {X  -159.990, Y  +457.497, Z    +0.000, E1  +334.597, E3 -454502.167}
SPL {X  -159.990, Y  +455.126, Z    +0.000, E1  +334.611, E3 -454512.775}
SPL {X  -159.990, Y  +453.438, Z    +0.000, E1  +334.615, E3 -454520.335}
SPL {X  -159.990, Y  +450.823, Z    +0.000, E1  +334.583, E3 -454531.955}
SPL {X  -159.990, Y  +446.894, Z    +0.000, E1  +334.572, E3 -454549.512}
SPL {X  -159.990, Y  +443.345, Z    +0.000, E1  +334.610, E3 -454565.519}
SPL {X  -159.990, Y  +441.077, Z    +0.000, E1  +334.631, E3 -454575.717}
SPL {X  -159.990, Y  +438.608, Z    +0.000, E1  +334.608, E3 -454586.714}
SPL {X  -159.990, Y  +434.852, Z    +0.000, E1  +334.585, E3 -454603.469}
SPL {X  -159.990, Y  +431.966, Z    +0.000, E1  +334.629, E3 -454616.466}
SPL {X  -159.990, Y  +429.079, Z    +0.000, E1  +334.593, E3 -454629.306}
SPL {X  -159.990, Y  +425.142, Z    +0.000, E1  +334.593, E3 -454646.909}
SPL {X  -159.990, Y  +421.010, Z    +0.000, E1  +334.582, E3 -454665.370}
SPL {X  -159.990, Y  +417.103, Z    +0.000, E1  +334.600, E3 -454682.873}
SPL {X  -159.990, Y  +414.457, Z    +0.000, E1  +334.626, E3 -454694.761}
SPL {X  -159.990, Y  +411.297, Z    +0.000, E1  +334.587, E3 -454708.818}
SPL {X  -159.990, Y  +407.450, Z    +0.000, E1  +334.599, E3 -454726.033}
SPL {X  -159.990, Y  +404.255, Z    +0.000, E1  +334.609, E3 -454740.323}
SPL {X  -159.990, Y  +401.103, Z    +0.000, E1  +334.596, E3 -454754.388}
SPL {X  -159.990, Y  +397.743, Z    +0.000, E1  +334.600, E3 -454769.438}
SPL {X  -159.990, Y  +394.848, Z    +0.000, E1  +334.621, E3 -454782.439}
SPL {X  -159.990, Y  +392.473, Z    +0.000, E1  +334.623, E3 -454793.066}
SPL {X  -159.990, Y  +390.187, Z    +0.000, E1  +334.622, E3 -454803.324}
SPL {X  -159.990, Y  +387.503, Z    +0.000, E1  +334.622, E3 -454815.319}
SPL {X  -159.990, Y  +384.711, Z    +0.000, E1  +334.612, E3 -454827.762}
SPL {X  -159.988, Y  +381.794, Z    +0.000, E1  +334.611, E3 -454840.797}
SPL {X  -159.958, Y  +379.279, Z    +0.000, E1  +334.625, E3 -454852.087}
SPL {X  -159.894, Y  +376.959, Z    +0.000, E1  +334.630, E3 -454862.532}
SPL {X  -159.765, Y  +374.027, Z    +0.000, E1  +334.633, E3 -454875.747}
SPL {X  -159.607, Y  +371.442, Z    +0.000, E1  +334.673, E3 -454887.522}
SPL {X  -159.379, Y  +368.534, Z    +0.000, E1  +334.684, E3 -454900.710}
SPL {X  -159.113, Y  +365.767, Z    +0.000, E1  +334.734, E3 -454913.350}
SPL {X  -158.798, Y  +363.007, Z    +0.000, E1  +334.761, E3 -454925.990}
SPL {X  -158.453, Y  +360.380, Z    +0.000, E1  +334.828, E3 -454938.134}
SPL {X  -158.127, Y  +358.155, Z    +0.000, E1  +334.874, E3 -454948.465}
SPL {X  -158.095, Y  +357.947, Z    +0.000, E1  +338.259, E3 -454980.037}
ENDSPLINE

SPLINE
SPL {X  -158.454, Y  +360.384, Z    +0.000, E1  +340.634, E3 -454992.189}
SPL {X  -159.737, Y  +373.507, Z    +0.000, E1  +349.689, E3 -455014.224}
SPL {X  -159.990, Y  +382.574, Z    +0.000, E1  +355.537, E3 -455020.912}
SPL {X  -159.990, Y  +389.909, Z    +0.000, E1  +360.662, E3 -455024.926}
SPL {X  -159.990, Y  +396.289, Z    +0.000, E1  +365.500, E3 -455028.706}
SPL {X  -159.990, Y  +407.941, Z    +0.000, E1  +374.126, E3 -455040.043}
SPL {X  -159.990, Y  +418.671, Z    +0.000, E1  +379.855, E3 -455059.460}
SPL {X  -159.990, Y  +429.878, Z    +0.000, E1  +383.330, E3 -455089.515}
SPL {X  -159.990, Y  +432.766, Z    +0.000, E1  +383.321, E3 -455103.737}
SPL {X  -159.990, Y  +435.585, Z    +0.000, E1  +383.327, E3 -455117.617}
SPL {X  -159.990, Y  +439.169, Z    +0.000, E1  +383.353, E3 -455135.200}
SPL {X  -159.990, Y  +442.945, Z    +0.000, E1  +383.339, E3 -455153.817}
SPL {X  -159.990, Y  +446.037, Z    +0.000, E1  +383.324, E3 -455169.067}
SPL {X  -159.990, Y  +448.341, Z    +0.000, E1  +383.317, E3 -455180.385}
SPL {X  -159.990, Y  +450.345, Z    +0.000, E1  +383.316, E3 -455190.263}
SPL {X  -159.990, Y  +452.828, Z    +0.000, E1  +383.330, E3 -455202.462}
SPL {X  -159.990, Y  +456.338, Z    +0.000, E1  +383.359, E3 -455219.655}
SPL {X  -159.990, Y  +459.480, Z    +0.000, E1  +383.323, E3 -455235.196}
SPL {X  -159.990, Y  +461.803, Z    +0.000, E1  +383.322, E3 -455246.631}
SPL {X  -159.990, Y  +464.971, Z    +0.000, E1  +383.357, E3 -455262.137}
SPL {X  -159.990, Y  +467.934, Z    +0.000, E1  +383.321, E3 -455276.794}
SPL {X  -159.990, Y  +469.939, Z    +0.000, E1  +383.319, E3 -455286.656}
SPL {X  -159.990, Y  +472.144, Z    +0.000, E1  +383.327, E3 -455297.507}
SPL {X  -159.990, Y  +474.152, Z    +0.000, E1  +383.309, E3 -455307.459}
SPL {X  -159.990, Y  +476.560, Z    +0.000, E1  +383.332, E3 -455319.267}
SPL {X  -159.990, Y  +478.770, Z    +0.000, E1  +383.306, E3 -455330.192}
SPL {X  -159.990, Y  +480.905, Z    +0.000, E1  +383.327, E3 -455340.660}
SPL {X  -159.990, Y  +484.251, Z    +0.000, E1  +383.352, E3 -455357.076}
SPL {X  -159.990, Y  +488.031, Z    +0.000, E1  +383.345, E3 -455375.708}
SPL {X  -159.990, Y  +491.121, Z    +0.000, E1  +383.323, E3 -455390.954}
SPL {X  -159.990, Y  +493.610, Z    +0.000, E1  +383.323, E3 -455403.207}
SPL {X  -159.990, Y  +496.863, Z    +0.000, E1  +383.350, E3 -455419.167}
SPL {X  -159.990, Y  +499.995, Z    +0.000, E1  +383.324, E3 -455434.628}
SPL {X  -159.990, Y  +502.341, Z    +0.000, E1  +383.320, E3 -455446.187}
SPL {X  -159.990, Y  +505.377, Z    +0.000, E1  +383.346, E3 -455461.078}
SPL {X  -159.990, Y  +508.697, Z    +0.000, E1  +383.335, E3 -455477.437}
SPL {X  -159.990, Y  +511.771, Z    +0.000, E1  +383.331, E3 -455492.584}
SPL {X  -159.990, Y  +514.016, Z    +0.000, E1  +383.308, E3 -455503.688}
SPL {X  -159.990, Y  +516.195, Z    +0.000, E1  +383.325, E3 -455514.376}
SPL {X  -159.990, Y  +518.925, Z    +0.000, E1  +383.333, E3 -455527.739}
SPL {X  -159.990, Y  +521.408, Z    +0.000, E1  +383.329, E3 -455539.948}
SPL {X  -159.990, Y  +523.942, Z    +0.000, E1  +383.333, E3 -455552.441}
SPL {X  -159.990, Y  +526.221, Z    +0.000, E1  +383.314, E3 -455563.717}
SPL {X  -159.990, Y  +527.834, Z    +0.000, E1  +383.311, E3 -455571.667}
SPL {X  -159.990, Y  +529.993, Z    +0.000, E1  +383.329, E3 -455582.243}
SPL {X  -159.990, Y  +532.441, Z    +0.000, E1  +383.322, E3 -455594.294}
SPL {X  -159.990, Y  +534.618, Z    +0.000, E1  +383.322, E3 -455605.027}
SPL {X  -159.990, Y  +537.024, Z    +0.000, E1  +383.321, E3 -455616.889}
SPL {X  -159.990, Y  +539.129, Z    +0.000, E1  +383.310, E3 -455627.272}
SPL {X  -159.990, Y  +541.183, Z    +0.000, E1  +383.319, E3 -455637.369}
SPL {X  -159.990, Y  +543.647, Z    +0.000, E1  +383.325, E3 -455649.472}
SPL {X  -159.990, Y  +545.957, Z    +0.000, E1  +383.318, E3 -455660.852}
SPL {X  -159.990, Y  +548.912, Z    +0.000, E1  +383.354, E3 -455675.311}
SPL {X  -159.990, Y  +551.655, Z    +0.000, E1  +383.320, E3 -455688.887}
SPL {X  -159.990, Y  +553.711, Z    +0.000, E1  +383.317, E3 -455699.008}
SPL {X  -159.990, Y  +556.481, Z    +0.000, E1  +383.354, E3 -455712.570}
SPL {X  -159.990, Y  +559.475, Z    +0.000, E1  +383.321, E3 -455727.376}
SPL {X  -159.990, Y  +561.830, Z    +0.000, E1  +383.325, E3 -455738.960}
SPL {X  -159.990, Y  +564.273, Z    +0.000, E1  +383.325, E3 -455750.984}
SPL {X  -159.990, Y  +566.342, Z    +0.000, E1  +383.314, E3 -455761.189}
SPL {X  -159.990, Y  +568.184, Z    +0.000, E1  +383.317, E3 -455770.250}
SPL {X  -159.990, Y  +570.314, Z    +0.000, E1  +383.326, E3 -455780.712}
SPL {X  -159.990, Y  +573.444, Z    +0.000, E1  +383.356, E3 -455796.052}
SPL {X  -159.990, Y  +576.445, Z    +0.000, E1  +383.320, E3 -455810.900}
SPL {X  -159.990, Y  +578.932, Z    +0.000, E1  +383.330, E3 -455823.117}
SPL {X  -159.990, Y  +581.497, Z    +0.000, E1  +383.329, E3 -455835.701}
SPL {X  -159.990, Y  +583.973, Z    +0.000, E1  +383.332, E3 -455847.886}
SPL {X  -159.990, Y  +586.020, Z    +0.000, E1  +383.323, E3 -455857.970}
SPL {X  -159.990, Y  +587.711, Z    +0.000, E1  +383.318, E3 -455866.310}
SPL {X  -159.990, Y  +589.763, Z    +0.000, E1  +383.328, E3 -455876.386}
SPL {X  -159.990, Y  +591.698, Z    +0.000, E1  +383.324, E3 -455885.871}
SPL {X  -159.990, Y  +593.847, Z    +0.000, E1  +383.340, E3 -455896.402}
SPL {X  -159.990, Y  +597.018, Z    +0.000, E1  +383.367, E3 -455911.934}
SPL {X  -159.990, Y  +599.887, Z    +0.000, E1  +383.341, E3 -455926.038}
SPL {X  -159.990, Y  +601.949, Z    +0.000, E1  +383.344, E3 -455936.165}
SPL {X  -159.990, Y  +605.106, Z    +0.000, E1  +383.383, E3 -455951.611}
SPL {X  -159.990, Y  +608.111, Z    +0.000, E1  +383.342, E3 -455966.462}
SPL {X  -159.990, Y  +610.073, Z    +0.000, E1  +383.343, E3 -455976.120}
SPL {X  -159.990, Y  +612.330, Z    +0.000, E1  +383.340, E3 -455987.247}
SPL {X  -159.990, Y  +615.036, Z    +0.000, E1  +383.353, E3 -456000.534}
SPL {X  -159.990, Y  +618.481, Z    +0.000, E1  +383.366, E3 -456017.472}
SPL {X  -159.990, Y  +621.517, Z    +0.000, E1  +383.337, E3 -456032.455}
SPL {X  -159.990, Y  +623.764, Z    +0.000, E1  +383.335, E3 -456043.506}
SPL {X  -159.990, Y  +626.608, Z    +0.000, E1  +383.361, E3 -456057.431}
SPL {X  -159.990, Y  +630.271, Z    +0.000, E1  +383.375, E3 -456075.392}
SPL {X  -159.990, Y  +633.318, Z    +0.000, E1  +383.339, E3 -456090.469}
SPL {X  -159.990, Y  +635.650, Z    +0.000, E1  +383.339, E3 -456101.940}
SPL {X  -159.990, Y  +638.406, Z    +0.000, E1  +383.354, E3 -456115.507}
SPL {X  -159.990, Y  +641.831, Z    +0.000, E1  +383.342, E3 -456132.454}
SPL {X  -159.990, Y  +644.884, Z    +0.000, E1  +383.324, E3 -456147.541}
SPL {X  -159.990, Y  +647.550, Z    +0.000, E1  +383.318, E3 -456160.708}
SPL {X  -159.990, Y  +650.790, Z    +0.000, E1  +383.346, E3 -456176.575}
SPL {X  -159.990, Y  +654.543, Z    +0.000, E1  +383.348, E3 -456195.028}
SPL {X  -159.990, Y  +658.319, Z    +0.000, E1  +383.349, E3 -456213.617}
SPL {X  -159.990, Y  +661.392, Z    +0.000, E1  +383.318, E3 -456228.820}
SPL {X  -159.990, Y  +663.662, Z    +0.000, E1  +383.322, E3 -456239.944}
SPL {X  -159.990, Y  +665.964, Z    +0.000, E1  +383.328, E3 -456251.235}
SPL {X  -159.990, Y  +667.870, Z    +0.000, E1  +383.320, E3 -456260.642}
SPL {X  -159.990, Y  +669.861, Z    +0.000, E1  +383.321, E3 -456270.443}
SPL {X  -159.990, Y  +671.893, Z    +0.000, E1  +383.319, E3 -456280.451}
SPL {X  -159.974, Y  +673.789, Z    +0.000, E1  +383.323, E3 -456289.767}
SPL {X  -159.924, Y  +676.110, Z    +0.000, E1  +383.320, E3 -456301.251}
SPL {X  -159.801, Y  +679.265, Z    +0.000, E1  +383.327, E3 -456316.870}
SPL {X  -159.626, Y  +682.287, Z    +0.000, E1  +383.280, E3 -456331.968}
SPL {X  -159.462, Y  +684.486, Z    +0.000, E1  +383.258, E3 -456342.968}
SPL {X  -159.212, Y  +687.262, Z    +0.000, E1  +383.238, E3 -456356.872}
SPL {X  -158.971, Y  +689.529, Z    +0.000, E1  +383.181, E3 -456368.332}
SPL {X  -158.658, Y  +692.098, Z    +0.000, E1  +383.176, E3 -456381.238}
ENDSPLINE

SPLINE
SPL {X  -159.063, Y  +688.696, Z    +0.000, E1  +377.094, E3 -456423.457}
SPL {X  -159.987, Y  +672.488, Z    +0.000, E1  +365.638, E3 -456447.522}
SPL {X  -159.990, Y  +663.928, Z    +0.000, E1  +359.662, E3 -456453.316}
SPL {X  -159.990, Y  +658.009, Z    +0.000, E1  +355.226, E3 -456457.016}
SPL {X  -159.990, Y  +651.879, Z    +0.000, E1  +350.548, E3 -456462.078}
SPL {X  -159.990, Y  +637.832, Z    +0.000, E1  +341.694, E3 -456479.670}
SPL {X  -159.990, Y  +626.634, Z    +0.000, E1  +337.968, E3 -456510.523}
SPL {X  -159.990, Y  +624.622, Z    +0.000, E1  +337.980, E3 -456521.106}
SPL {X  -159.990, Y  +622.489, Z    +0.000, E1  +337.969, E3 -456532.273}
SPL {X  -159.990, Y  +619.267, Z    +0.000, E1  +337.938, E3 -456549.107}
SPL {X  -159.990, Y  +615.467, Z    +0.000, E1  +337.940, E3 -456569.043}
SPL {X  -159.990, Y  +612.600, Z    +0.000, E1  +337.975, E3 -456584.154}
SPL {X  -159.990, Y  +610.646, Z    +0.000, E1  +337.979, E3 -456594.411}
SPL {X  -159.990, Y  +608.810, Z    +0.000, E1  +337.977, E3 -456604.044}
SPL {X  -159.990, Y  +606.481, Z    +0.000, E1  +337.967, E3 -456616.220}
SPL {X  -159.990, Y  +603.419, Z    +0.000, E1  +337.936, E3 -456632.159}
SPL {X  -159.990, Y  +600.642, Z    +0.000, E1  +337.968, E3 -456646.789}
SPL {X  -159.990, Y  +598.568, Z    +0.000, E1  +337.954, E3 -456657.581}
SPL {X  -159.990, Y  +595.493, Z    +0.000, E1  +337.930, E3 -456673.665}
SPL {X  -159.990, Y  +592.865, Z    +0.000, E1  +337.964, E3 -456687.493}
SPL {X  -159.990, Y  +590.803, Z    +0.000, E1  +337.954, E3 -456698.284}
SPL {X  -159.990, Y  +588.288, Z    +0.000, E1  +337.950, E3 -456711.448}
SPL {X  -159.990, Y  +586.040, Z    +0.000, E1  +337.954, E3 -456723.193}
SPL {X  -159.990, Y  +584.080, Z    +0.000, E1  +337.953, E3 -456733.453}
SPL {X  -159.990, Y  +581.924, Z    +0.000, E1  +337.949, E3 -456744.753}
SPL {X  -159.990, Y  +579.673, Z    +0.000, E1  +337.950, E3 -456756.552}
SPL {X  -159.990, Y  +576.961, Z    +0.000, E1  +337.936, E3 -456770.731}
SPL {X  -159.990, Y  +574.188, Z    +0.000, E1  +337.947, E3 -456785.278}
SPL {X  -159.990, Y  +571.954, Z    +0.000, E1  +337.959, E3 -456797.036}
SPL {X  -159.990, Y  +570.110, Z    +0.000, E1  +337.958, E3 -456806.686}
SPL {X  -159.990, Y  +568.165, Z    +0.000, E1  +337.957, E3 -456816.866}
SPL {X  -159.990, Y  +565.292, Z    +0.000, E1  +337.922, E3 -456831.844}
SPL {X  -159.990, Y  +562.598, Z    +0.000, E1  +337.958, E3 -456846.055}
SPL {X  -159.990, Y  +560.652, Z    +0.000, E1  +337.962, E3 -456856.267}
SPL {X  -159.990, Y  +558.143, Z    +0.000, E1  +337.928, E3 -456869.299}
SPL {X  -159.990, Y  +555.329, Z    +0.000, E1  +337.943, E3 -456884.043}
SPL {X  -159.990, Y  +553.115, Z    +0.000, E1  +337.946, E3 -456895.649}
SPL {X  -159.990, Y  +550.886, Z    +0.000, E1  +337.944, E3 -456907.330}
SPL {X  -159.990, Y  +548.568, Z    +0.000, E1  +337.944, E3 -456919.451}
SPL {X  -159.990, Y  +546.537, Z    +0.000, E1  +337.948, E3 -456930.086}
SPL {X  -159.990, Y  +545.062, Z    +0.000, E1  +337.955, E3 -456937.845}
SPL {X  -159.990, Y  +543.060, Z    +0.000, E1  +337.943, E3 -456948.324}
SPL {X  -159.990, Y  +539.928, Z    +0.000, E1  +337.917, E3 -456964.665}
SPL {X  -159.990, Y  +536.935, Z    +0.000, E1  +337.942, E3 -456980.382}
SPL {X  -159.990, Y  +534.656, Z    +0.000, E1  +337.946, E3 -456992.326}
SPL {X  -159.990, Y  +532.453, Z    +0.000, E1  +337.944, E3 -457003.853}
SPL {X  -159.990, Y  +530.660, Z    +0.000, E1  +337.952, E3 -457013.256}
SPL {X  -159.990, Y  +528.702, Z    +0.000, E1  +337.939, E3 -457023.469}
SPL {X  -159.990, Y  +525.760, Z    +0.000, E1  +337.914, E3 -457038.810}
SPL {X  -159.990, Y  +522.838, Z    +0.000, E1  +337.933, E3 -457054.177}
SPL {X  -159.990, Y  +520.708, Z    +0.000, E1  +337.953, E3 -457065.370}
SPL {X  -159.990, Y  +518.216, Z    +0.000, E1  +337.909, E3 -457078.287}
SPL {X  -159.990, Y  +515.568, Z    +0.000, E1  +338.084, E3 -457093.517}
ENDSPLINE

SPLINE
SPL {X  -159.990, Y  +518.374, Z    +0.000, E1  +341.240, E3 -457106.104}
ENDSPLINE

SPLINE
SPL {X  -159.990, Y  +513.606, Z    +0.000, E1  +339.879, E3 -457122.015}
SPL {X  -159.990, Y  +508.660, Z    +0.000, E1  +338.515, E3 -457137.444}
SPL {X  -159.990, Y  +505.237, Z    +0.000, E1  +337.606, E3 -457147.702}
SPL {X  -159.990, Y  +501.963, Z    +0.000, E1  +336.712, E3 -457156.805}
SPL {X  -159.990, Y  +498.406, Z    +0.000, E1  +335.789, E3 -457166.556}
SPL {X  -159.990, Y  +494.693, Z    +0.000, E1  +334.929, E3 -457177.024}
SPL {X  -159.990, Y  +491.649, Z    +0.000, E1  +334.596, E3 -457188.226}
SPL {X  -159.990, Y  +488.807, Z    +0.000, E1  +334.603, E3 -457200.951}
SPL {X  -159.990, Y  +486.070, Z    +0.000, E1  +334.601, E3 -457213.182}
SPL {X  -159.990, Y  +483.747, Z    +0.000, E1  +334.616, E3 -457223.595}
SPL {X  -159.990, Y  +481.980, Z    +0.000, E1  +334.616, E3 -457231.492}
SPL {X  -159.990, Y  +479.252, Z    +0.000, E1  +334.588, E3 -457243.634}
SPL {X  -159.990, Y  +475.940, Z    +0.000, E1  +334.597, E3 -457258.454}
SPL {X  -159.990, Y  +473.026, Z    +0.000, E1  +334.601, E3 -457271.484}
SPL {X  -159.990, Y  +470.047, Z    +0.000, E1  +334.598, E3 -457284.802}
SPL {X  -159.990, Y  +466.213, Z    +0.000, E1  +334.567, E3 -457301.882}
SPL {X  -159.990, Y  +462.520, Z    +0.000, E1  +334.600, E3 -457318.451}
SPL {X  -159.990, Y  +460.081, Z    +0.000, E1  +334.610, E3 -457329.352}
SPL {X  -159.990, Y  +457.497, Z    +0.000, E1  +334.597, E3 -457340.876}
SPL {X  -159.990, Y  +455.126, Z    +0.000, E1  +334.611, E3 -457351.485}
SPL {X  -159.990, Y  +452.123, Z    +0.000, E1  +334.574, E3 -457364.842}
SPL {X  -159.990, Y  +448.503, Z    +0.000, E1  +334.590, E3 -457381.044}
SPL {X  -159.990, Y  +445.882, Z    +0.000, E1  +334.615, E3 -457392.846}
SPL {X  -159.990, Y  +443.345, Z    +0.000, E1  +334.610, E3 -457404.229}
SPL {X  -159.990, Y  +441.077, Z    +0.000, E1  +334.631, E3 -457414.427}
SPL {X  -159.990, Y  +438.608, Z    +0.000, E1  +334.608, E3 -457425.424}
SPL {X  -159.990, Y  +434.852, Z    +0.000, E1  +334.585, E3 -457442.178}
SPL {X  -159.990, Y  +430.645, Z    +0.000, E1  +334.586, E3 -457460.998}
SPL {X  -159.990, Y  +426.865, Z    +0.000, E1  +334.602, E3 -457477.927}
SPL {X  -159.990, Y  +424.251, Z    +0.000, E1  +334.625, E3 -457489.664}
SPL {X  -159.990, Y  +421.010, Z    +0.000, E1  +334.582, E3 -457504.079}
SPL {X  -159.990, Y  +417.103, Z    +0.000, E1  +334.600, E3 -457521.583}
SPL {X  -159.990, Y  +413.684, Z    +0.000, E1  +334.603, E3 -457536.882}
SPL {X  -159.990, Y  +410.645, Z    +0.000, E1  +334.615, E3 -457550.494}
SPL {X  -159.990, Y  +407.450, Z    +0.000, E1  +334.599, E3 -457564.742}
SPL {X  -159.990, Y  +403.513, Z    +0.000, E1  +334.580, E3 -457582.296}
SPL {X  -159.990, Y  +399.294, Z    +0.000, E1  +334.582, E3 -457601.176}
SPL {X  -159.990, Y  +395.411, Z    +0.000, E1  +334.600, E3 -457618.590}
SPL {X  -159.990, Y  +392.473, Z    +0.000, E1  +334.623, E3 -457631.775}
SPL {X  -159.990, Y  +390.187, Z    +0.000, E1  +334.622, E3 -457642.033}
SPL {X  -159.990, Y  +387.503, Z    +0.000, E1  +334.622, E3 -457654.028}
SPL {X  -159.990, Y  +384.711, Z    +0.000, E1  +334.612, E3 -457666.472}
SPL {X  -159.988, Y  +381.794, Z    +0.000, E1  +334.611, E3 -457679.507}
SPL {X  -159.958, Y  +379.279, Z    +0.000, E1  +334.625, E3 -457690.797}
SPL {X  -159.894, Y  +376.959, Z    +0.000, E1  +334.630, E3 -457701.241}
SPL {X  -159.765, Y  +374.027, Z    +0.000, E1  +334.633, E3 -457714.457}
SPL {X  -159.607, Y  +371.442, Z    +0.000, E1  +334.673, E3 -457726.232}
SPL {X  -159.379, Y  +368.534, Z    +0.000, E1  +334.684, E3 -457739.420}
SPL {X  -159.113, Y  +365.767, Z    +0.000, E1  +334.734, E3 -457752.059}
SPL {X  -158.798, Y  +363.007, Z    +0.000, E1  +334.761, E3 -457764.699}
SPL {X  -158.453, Y  +360.380, Z    +0.000, E1  +334.828, E3 -457776.844}
SPL {X  -158.127, Y  +358.155, Z    +0.000, E1  +334.874, E3 -457787.175}
SPL {X  -158.095, Y  +357.947, Z    +0.000, E1  +338.259, E3 -457818.747}
ENDSPLINE

SPLINE
SPL {X  -158.454, Y  +360.384, Z    +0.000, E1  +340.634, E3 -457830.898}
SPL {X  -159.737, Y  +373.507, Z    +0.000, E1  +349.689, E3 -457852.934}
SPL {X  -159.990, Y  +382.574, Z    +0.000, E1  +355.537, E3 -457859.621}
SPL {X  -159.990, Y  +387.496, Z    +0.000, E1  +358.996, E3 -457862.366}
SPL {X  -159.990, Y  +395.121, Z    +0.000, E1  +364.514, E3 -457866.679}
SPL {X  -159.990, Y  +407.941, Z    +0.000, E1  +374.126, E3 -457878.753}
SPL {X  -159.990, Y  +418.671, Z    +0.000, E1  +379.855, E3 -457898.169}
SPL {X  -159.990, Y  +429.878, Z    +0.000, E1  +383.330, E3 -457928.224}
SPL {X  -159.990, Y  +432.766, Z    +0.000, E1  +383.321, E3 -457942.447}
SPL {X  -159.990, Y  +434.794, Z    +0.000, E1  +383.304, E3 -457952.478}
SPL {X  -159.990, Y  +437.007, Z    +0.000, E1  +383.323, E3 -457963.331}
SPL {X  -159.990, Y  +439.778, Z    +0.000, E1  +383.323, E3 -457976.963}
SPL {X  -159.990, Y  +442.010, Z    +0.000, E1  +383.308, E3 -457987.984}
SPL {X  -159.990, Y  +443.729, Z    +0.000, E1  +383.310, E3 -457996.440}
SPL {X  -159.990, Y  +446.037, Z    +0.000, E1  +383.324, E3 -458007.777}
SPL {X  -159.990, Y  +448.341, Z    +0.000, E1  +383.317, E3 -458019.095}
SPL {X  -159.990, Y  +450.345, Z    +0.000, E1  +383.316, E3 -458028.973}
SPL {X  -159.990, Y  +452.828, Z    +0.000, E1  +383.330, E3 -458041.172}
SPL {X  -159.990, Y  +455.244, Z    +0.000, E1  +383.317, E3 -458053.072}
SPL {X  -159.990, Y  +457.167, Z    +0.000, E1  +383.324, E3 -458062.502}
SPL {X  -159.990, Y  +459.480, Z    +0.000, E1  +383.323, E3 -458073.906}
SPL {X  -159.990, Y  +462.520, Z    +0.000, E1  +383.350, E3 -458088.810}
SPL {X  -159.990, Y  +465.602, Z    +0.000, E1  +383.328, E3 -458104.010}
SPL {X  -159.990, Y  +467.934, Z    +0.000, E1  +383.321, E3 -458115.504}
SPL {X  -159.990, Y  +469.939, Z    +0.000, E1  +383.319, E3 -458125.366}
SPL {X  -159.990, Y  +472.144, Z    +0.000, E1  +383.327, E3 -458136.216}
SPL {X  -159.990, Y  +474.152, Z    +0.000, E1  +383.309, E3 -458146.168}
SPL {X  -159.990, Y  +476.560, Z    +0.000, E1  +383.332, E3 -458157.977}
SPL {X  -159.990, Y  +478.770, Z    +0.000, E1  +383.306, E3 -458168.902}
SPL {X  -159.990, Y  +480.905, Z    +0.000, E1  +383.327, E3 -458179.370}
SPL {X  -159.990, Y  +484.251, Z    +0.000, E1  +383.352, E3 -458195.785}
SPL {X  -159.990, Y  +488.031, Z    +0.000, E1  +383.345, E3 -458214.418}
SPL {X  -159.990, Y  +491.121, Z    +0.000, E1  +383.323, E3 -458229.664}
SPL {X  -159.990, Y  +493.610, Z    +0.000, E1  +383.323, E3 -458241.917}
SPL {X  -159.990, Y  +495.794, Z    +0.000, E1  +383.312, E3 -458252.690}
SPL {X  -159.990, Y  +497.668, Z    +0.000, E1  +383.317, E3 -458261.900}
SPL {X  -159.990, Y  +499.995, Z    +0.000, E1  +383.324, E3 -458273.338}
SPL {X  -159.990, Y  +502.341, Z    +0.000, E1  +383.320, E3 -458284.897}
SPL {X  -159.990, Y  +504.419, Z    +0.000, E1  +383.313, E3 -458295.139}
SPL {X  -159.990, Y  +507.187, Z    +0.000, E1  +383.346, E3 -458308.692}
SPL {X  -159.990, Y  +510.344, Z    +0.000, E1  +383.327, E3 -458324.277}
SPL {X  -159.990, Y  +512.484, Z    +0.000, E1  +383.309, E3 -458334.849}
SPL {X  -159.990, Y  +514.016, Z    +0.000, E1  +383.308, E3 -458342.398}
SPL {X  -159.990, Y  +516.195, Z    +0.000, E1  +383.325, E3 -458353.086}
SPL {X  -159.990, Y  +518.925, Z    +0.000, E1  +383.333, E3 -458366.449}
SPL {X  -159.990, Y  +521.408, Z    +0.000, E1  +383.329, E3 -458378.658}
SPL {X  -159.990, Y  +523.942, Z    +0.000, E1  +383.333, E3 -458391.151}
SPL {X  -159.990, Y  +527.007, Z    +0.000, E1  +383.339, E3 -458406.250}
SPL {X  -159.990, Y  +529.993, Z    +0.000, E1  +383.329, E3 -458420.953}
SPL {X  -159.990, Y  +532.441, Z    +0.000, E1  +383.322, E3 -458433.003}
SPL {X  -159.990, Y  +534.618, Z    +0.000, E1  +383.322, E3 -458443.737}
SPL {X  -159.990, Y  +537.024, Z    +0.000, E1  +383.321, E3 -458455.599}
SPL {X  -159.990, Y  +539.129, Z    +0.000, E1  +383.310, E3 -458465.982}
SPL {X  -159.990, Y  +541.183, Z    +0.000, E1  +383.319, E3 -458476.079}
SPL {X  -159.990, Y  +543.647, Z    +0.000, E1  +383.325, E3 -458488.182}
SPL {X  -159.990, Y  +545.957, Z    +0.000, E1  +383.318, E3 -458499.561}
SPL {X  -159.990, Y  +548.912, Z    +0.000, E1  +383.354, E3 -458514.021}
SPL {X  -159.990, Y  +551.655, Z    +0.000, E1  +383.320, E3 -458527.596}
SPL {X  -159.990, Y  +553.711, Z    +0.000, E1  +383.317, E3 -458537.718}
SPL {X  -159.990, Y  +556.481, Z    +0.000, E1  +383.354, E3 -458551.280}
SPL {X  -159.990, Y  +559.475, Z    +0.000, E1  +383.321, E3 -458566.085}
SPL {X  -159.990, Y  +561.830, Z    +0.000, E1  +383.325, E3 -458577.670}
SPL {X  -159.990, Y  +564.273, Z    +0.000, E1  +383.325, E3 -458589.694}
SPL {X  -159.990, Y  +567.351, Z    +0.000, E1  +383.348, E3 -458604.790}
SPL {X  -159.990, Y  +570.314, Z    +0.000, E1  +383.326, E3 -458619.422}
SPL {X  -159.990, Y  +572.504, Z    +0.000, E1  +383.321, E3 -458630.207}
SPL {X  -159.990, Y  +575.653, Z    +0.000, E1  +383.355, E3 -458645.644}
SPL {X  -159.990, Y  +578.932, Z    +0.000, E1  +383.330, E3 -458661.826}
SPL {X  -159.990, Y  +581.497, Z    +0.000, E1  +383.329, E3 -458674.411}
SPL {X  -159.990, Y  +583.973, Z    +0.000, E1  +383.332, E3 -458686.596}
SPL {X  -159.990, Y  +586.020, Z    +0.000, E1  +383.323, E3 -458696.680}
SPL {X  -159.990, Y  +587.711, Z    +0.000, E1  +383.318, E3 -458705.020}
SPL {X  -159.990, Y  +589.763, Z    +0.000, E1  +383.328, E3 -458715.096}
SPL {X  -159.990, Y  +591.698, Z    +0.000, E1  +383.324, E3 -458724.581}
SPL {X  -159.990, Y  +593.847, Z    +0.000, E1  +383.340, E3 -458735.111}
SPL {X  -159.990, Y  +597.018, Z    +0.000, E1  +383.367, E3 -458750.643}
SPL {X  -159.990, Y  +599.887, Z    +0.000, E1  +383.341, E3 -458764.748}
SPL {X  -159.990, Y  +601.949, Z    +0.000, E1  +383.344, E3 -458774.874}
SPL {X  -159.990, Y  +605.106, Z    +0.000, E1  +383.383, E3 -458790.320}
SPL {X  -159.990, Y  +608.111, Z    +0.000, E1  +383.342, E3 -458805.171}
SPL {X  -159.990, Y  +610.073, Z    +0.000, E1  +383.343, E3 -458814.829}
SPL {X  -159.990, Y  +613.021, Z    +0.000, E1  +383.365, E3 -458829.300}
SPL {X  -159.990, Y  +615.657, Z    +0.000, E1  +383.331, E3 -458842.348}
SPL {X  -159.990, Y  +617.658, Z    +0.000, E1  +383.335, E3 -458852.190}
SPL {X  -159.990, Y  +620.788, Z    +0.000, E1  +383.368, E3 -458867.523}
SPL {X  -159.990, Y  +624.347, Z    +0.000, E1  +383.355, E3 -458885.044}
SPL {X  -159.990, Y  +627.144, Z    +0.000, E1  +383.340, E3 -458898.813}
SPL {X  -159.990, Y  +630.271, Z    +0.000, E1  +383.375, E3 -458914.102}
SPL {X  -159.990, Y  +633.318, Z    +0.000, E1  +383.339, E3 -458929.179}
SPL {X  -159.990, Y  +635.650, Z    +0.000, E1  +383.339, E3 -458940.650}
SPL {X  -159.990, Y  +638.406, Z    +0.000, E1  +383.354, E3 -458954.217}
SPL {X  -159.990, Y  +641.831, Z    +0.000, E1  +383.342, E3 -458971.164}
SPL {X  -159.990, Y  +644.884, Z    +0.000, E1  +383.324, E3 -458986.251}
SPL {X  -159.990, Y  +647.550, Z    +0.000, E1  +383.318, E3 -458999.418}
SPL {X  -159.990, Y  +650.790, Z    +0.000, E1  +383.346, E3 -459015.284}
SPL {X  -159.990, Y  +654.543, Z    +0.000, E1  +383.348, E3 -459033.737}
SPL {X  -159.990, Y  +658.319, Z    +0.000, E1  +383.349, E3 -459052.327}
SPL {X  -159.990, Y  +661.392, Z    +0.000, E1  +383.318, E3 -459067.530}
SPL {X  -159.990, Y  +663.662, Z    +0.000, E1  +383.322, E3 -459078.654}
SPL {X  -159.990, Y  +665.964, Z    +0.000, E1  +383.328, E3 -459089.945}
SPL {X  -159.990, Y  +668.989, Z    +0.000, E1  +383.359, E3 -459104.780}
SPL {X  -159.983, Y  +672.946, Z    +0.000, E1  +383.359, E3 -459124.262}
SPL {X  -159.924, Y  +676.110, Z    +0.000, E1  +383.320, E3 -459139.961}
SPL {X  -159.845, Y  +678.302, Z    +0.000, E1  +383.298, E3 -459150.863}
SPL {X  -159.760, Y  +680.081, Z    +0.000, E1  +383.288, E3 -459159.706}
SPL {X  -159.626, Y  +682.287, Z    +0.000, E1  +383.280, E3 -459170.678}
SPL {X  -159.462, Y  +684.486, Z    +0.000, E1  +383.258, E3 -459181.678}
SPL {X  -159.212, Y  +687.262, Z    +0.000, E1  +383.238, E3 -459195.581}
SPL {X  -158.971, Y  +689.529, Z    +0.000, E1  +383.181, E3 -459207.041}
SPL {X  -158.658, Y  +692.098, Z    +0.000, E1  +383.176, E3 -459219.948}
ENDSPLINE

SPLINE
SPL {X  -159.063, Y  +688.696, Z    +0.000, E1  +377.094, E3 -459262.166}
SPL {X  -159.987, Y  +672.488, Z    +0.000, E1  +365.638, E3 -459286.231}
SPL {X  -159.990, Y  +663.928, Z    +0.000, E1  +359.662, E3 -459292.026}
SPL {X  -159.990, Y  +658.009, Z    +0.000, E1  +355.226, E3 -459295.726}
SPL {X  -159.990, Y  +651.879, Z    +0.000, E1  +350.548, E3 -459300.788}
SPL {X  -159.990, Y  +637.832, Z    +0.000, E1  +341.694, E3 -459318.379}
SPL {X  -159.990, Y  +626.634, Z    +0.000, E1  +337.968, E3 -459349.232}
SPL {X  -159.990, Y  +624.622, Z    +0.000, E1  +337.980, E3 -459359.816}
SPL {X  -159.990, Y  +622.489, Z    +0.000, E1  +337.969, E3 -459370.982}
SPL {X  -159.990, Y  +619.955, Z    +0.000, E1  +337.968, E3 -459384.272}
SPL {X  -159.990, Y  +617.386, Z    +0.000, E1  +337.968, E3 -459397.747}
SPL {X  -159.990, Y  +614.863, Z    +0.000, E1  +337.969, E3 -459410.979}
SPL {X  -159.990, Y  +612.600, Z    +0.000, E1  +337.975, E3 -459422.863}
SPL {X  -159.990, Y  +610.646, Z    +0.000, E1  +337.979, E3 -459433.121}
SPL {X  -159.990, Y  +608.810, Z    +0.000, E1  +337.977, E3 -459442.754}
SPL {X  -159.990, Y  +605.804, Z    +0.000, E1  +337.936, E3 -459458.399}
SPL {X  -159.990, Y  +602.819, Z    +0.000, E1  +337.963, E3 -459474.070}
SPL {X  -159.990, Y  +600.642, Z    +0.000, E1  +337.968, E3 -459485.498}
SPL {X  -159.990, Y  +598.568, Z    +0.000, E1  +337.954, E3 -459496.291}
SPL {X  -159.990, Y  +596.440, Z    +0.000, E1  +337.964, E3 -459507.473}
SPL {X  -159.990, Y  +593.768, Z    +0.000, E1  +337.929, E3 -459521.406}
SPL {X  -159.990, Y  +590.068, Z    +0.000, E1  +337.924, E3 -459540.774}
SPL {X  -159.990, Y  +586.620, Z    +0.000, E1  +337.935, E3 -459558.836}
SPL {X  -159.990, Y  +584.080, Z    +0.000, E1  +337.953, E3 -459572.163}
SPL {X  -159.990, Y  +581.924, Z    +0.000, E1  +337.949, E3 -459583.463}
SPL {X  -159.990, Y  +579.673, Z    +0.000, E1  +337.950, E3 -459595.261}
SPL {X  -159.990, Y  +576.961, Z    +0.000, E1  +337.936, E3 -459609.441}
SPL {X  -159.990, Y  +574.188, Z    +0.000, E1  +337.947, E3 -459623.988}
SPL {X  -159.990, Y  +571.954, Z    +0.000, E1  +337.959, E3 -459635.746}
SPL {X  -159.990, Y  +570.110, Z    +0.000, E1  +337.958, E3 -459645.396}
SPL {X  -159.990, Y  +568.165, Z    +0.000, E1  +337.957, E3 -459655.576}
SPL {X  -159.990, Y  +565.292, Z    +0.000, E1  +337.922, E3 -459670.554}
SPL {X  -159.990, Y  +562.598, Z    +0.000, E1  +337.958, E3 -459684.765}
SPL {X  -159.990, Y  +560.652, Z    +0.000, E1  +337.962, E3 -459694.977}
SPL {X  -159.990, Y  +558.143, Z    +0.000, E1  +337.928, E3 -459708.009}
SPL {X  -159.990, Y  +555.329, Z    +0.000, E1  +337.943, E3 -459722.753}
SPL {X  -159.990, Y  +553.115, Z    +0.000, E1  +337.946, E3 -459734.358}
SPL {X  -159.990, Y  +550.886, Z    +0.000, E1  +337.944, E3 -459746.040}
SPL {X  -159.990, Y  +548.568, Z    +0.000, E1  +337.944, E3 -459758.161}
SPL {X  -159.990, Y  +546.537, Z    +0.000, E1  +337.948, E3 -459768.796}
SPL {X  -159.990, Y  +545.062, Z    +0.000, E1  +337.955, E3 -459776.554}
SPL {X  -159.990, Y  +543.060, Z    +0.000, E1  +337.943, E3 -459787.034}
SPL {X  -159.990, Y  +539.928, Z    +0.000, E1  +337.917, E3 -459803.375}
SPL {X  -159.990, Y  +536.935, Z    +0.000, E1  +337.942, E3 -459819.092}
SPL {X  -159.990, Y  +534.656, Z    +0.000, E1  +337.946, E3 -459831.036}
SPL {X  -159.990, Y  +531.679, Z    +0.000, E1  +337.913, E3 -459846.550}
SPL {X  -159.990, Y  +527.941, Z    +0.000, E1  +337.907, E3 -459866.092}
SPL {X  -159.990, Y  +525.053, Z    +0.000, E1  +337.942, E3 -459881.282}
SPL {X  -159.990, Y  +522.838, Z    +0.000, E1  +337.933, E3 -459892.886}
SPL {X  -159.990, Y  +519.698, Z    +0.000, E1  +337.916, E3 -459909.269}
SPL {X  -159.990, Y  +517.251, Z    +0.000, E1  +337.946, E3 -459922.129}
SPL {X  -159.990, Y  +515.568, Z    +0.000, E1  +338.084, E3 -459932.226}
ENDSPLINE

SPLINE
SPL {X  -159.990, Y  +517.293, Z    +0.000, E1  +340.923, E3 -459948.525}
ENDSPLINE

SPLINE
SPL {X  -159.990, Y  +512.548, Z    +0.000, E1  +339.587, E3 -459964.100}
SPL {X  -159.990, Y  +508.660, Z    +0.000, E1  +338.515, E3 -459976.154}
SPL {X  -159.990, Y  +503.499, Z    +0.000, E1  +337.116, E3 -459991.233}
SPL {X  -159.990, Y  +498.406, Z    +0.000, E1  +335.789, E3 -460005.266}
SPL {X  -159.990, Y  +494.693, Z    +0.000, E1  +334.929, E3 -460015.733}
SPL {X  -159.990, Y  +491.649, Z    +0.000, E1  +334.596, E3 -460026.936}
SPL {X  -159.990, Y  +488.807, Z    +0.000, E1  +334.603, E3 -460039.660}
SPL {X  -159.990, Y  +486.070, Z    +0.000, E1  +334.601, E3 -460051.891}
SPL {X  -159.990, Y  +482.821, Z    +0.000, E1  +334.589, E3 -460066.393}
SPL {X  -159.990, Y  +480.183, Z    +0.000, E1  +334.616, E3 -460078.233}
SPL {X  -159.990, Y  +477.508, Z    +0.000, E1  +334.590, E3 -460090.142}
SPL {X  -159.990, Y  +473.634, Z    +0.000, E1  +334.574, E3 -460107.431}
SPL {X  -159.990, Y  +470.047, Z    +0.000, E1  +334.598, E3 -460123.512}
SPL {X  -159.990, Y  +467.082, Z    +0.000, E1  +334.601, E3 -460136.759}
SPL {X  -159.990, Y  +464.063, Z    +0.000, E1  +334.595, E3 -460150.254}
SPL {X  -159.990, Y  +460.712, Z    +0.000, E1  +334.589, E3 -460165.214}
SPL {X  -159.990, Y  +457.497, Z    +0.000, E1  +334.597, E3 -460179.586}
SPL {X  -159.990, Y  +454.323, Z    +0.000, E1  +334.588, E3 -460193.745}
SPL {X  -159.990, Y  +450.823, Z    +0.000, E1  +334.583, E3 -460209.374}
SPL {X  -159.990, Y  +447.982, Z    +0.000, E1  +334.607, E3 -460222.115}
SPL {X  -159.990, Y  +445.108, Z    +0.000, E1  +334.593, E3 -460234.992}
SPL {X  -159.990, Y  +441.797, Z    +0.000, E1  +334.610, E3 -460249.871}
SPL {X  -159.990, Y  +439.442, Z    +0.000, E1  +334.631, E3 -460260.448}
SPL {X  -159.990, Y  +436.316, Z    +0.000, E1  +334.580, E3 -460274.330}
SPL {X  -159.990, Y  +432.613, Z    +0.000, E1  +334.610, E3 -460290.955}
SPL {X  -159.990, Y  +429.827, Z    +0.000, E1  +334.620, E3 -460303.432}
SPL {X  -159.990, Y  +426.865, Z    +0.000, E1  +334.602, E3 -460316.637}
SPL {X  -159.990, Y  +423.417, Z    +0.000, E1  +334.600, E3 -460332.053}
SPL {X  -159.990, Y  +420.283, Z    +0.000, E1  +334.614, E3 -460346.097}
SPL {X  -159.990, Y  +417.103, Z    +0.000, E1  +334.600, E3 -460360.292}
SPL {X  -159.990, Y  +413.684, Z    +0.000, E1  +334.603, E3 -460375.592}
SPL {X  -159.990, Y  +410.645, Z    +0.000, E1  +334.615, E3 -460389.204}
SPL {X  -159.990, Y  +407.450, Z    +0.000, E1  +334.599, E3 -460403.452}
SPL {X  -159.990, Y  +403.513, Z    +0.000, E1  +334.580, E3 -460421.006}
SPL {X  -159.990, Y  +399.294, Z    +0.000, E1  +334.582, E3 -460439.885}
SPL {X  -159.990, Y  +395.411, Z    +0.000, E1  +334.600, E3 -460457.300}
SPL {X  -159.990, Y  +392.473, Z    +0.000, E1  +334.623, E3 -460470.485}
SPL {X  -159.990, Y  +390.187, Z    +0.000, E1  +334.622, E3 -460480.743}
SPL {X  -159.990, Y  +387.503, Z    +0.000, E1  +334.622, E3 -460492.738}
SPL {X  -159.990, Y  +384.711, Z    +0.000, E1  +334.612, E3 -460505.182}
SPL {X  -159.988, Y  +381.794, Z    +0.000, E1  +334.611, E3 -460518.217}
SPL {X  -159.958, Y  +379.279, Z    +0.000, E1  +334.625, E3 -460529.507}
SPL {X  -159.894, Y  +376.959, Z    +0.000, E1  +334.630, E3 -460539.951}
SPL {X  -159.765, Y  +374.027, Z    +0.000, E1  +334.633, E3 -460553.167}
SPL {X  -159.607, Y  +371.442, Z    +0.000, E1  +334.673, E3 -460564.942}
SPL {X  -159.379, Y  +368.534, Z    +0.000, E1  +334.684, E3 -460578.129}
SPL {X  -159.113, Y  +365.767, Z    +0.000, E1  +334.734, E3 -460590.769}
SPL {X  -158.798, Y  +363.007, Z    +0.000, E1  +334.761, E3 -460603.409}
SPL {X  -158.453, Y  +360.380, Z    +0.000, E1  +334.828, E3 -460615.554}
SPL {X  -158.127, Y  +358.155, Z    +0.000, E1  +334.874, E3 -460625.884}
SPL {X  -158.095, Y  +357.947, Z    +0.000, E1  +338.259, E3 -460657.457}
ENDSPLINE

SPLINE
SPL {X  -158.454, Y  +360.384, Z    +0.000, E1  +340.634, E3 -460669.608}
SPL {X  -159.737, Y  +373.507, Z    +0.000, E1  +349.689, E3 -460691.643}
SPL {X  -159.990, Y  +382.574, Z    +0.000, E1  +355.537, E3 -460698.331}
SPL {X  -159.990, Y  +389.909, Z    +0.000, E1  +360.662, E3 -460702.346}
SPL {X  -159.990, Y  +396.289, Z    +0.000, E1  +365.500, E3 -460706.126}
SPL {X  -159.990, Y  +407.941, Z    +0.000, E1  +374.126, E3 -460717.463}
SPL {X  -159.990, Y  +418.671, Z    +0.000, E1  +379.855, E3 -460736.879}
SPL {X  -159.990, Y  +429.878, Z    +0.000, E1  +383.330, E3 -460766.934}
SPL {X  -159.990, Y  +432.766, Z    +0.000, E1  +383.321, E3 -460781.156}
SPL {X  -159.990, Y  +434.794, Z    +0.000, E1  +383.304, E3 -460791.188}
SPL {X  -159.990, Y  +437.007, Z    +0.000, E1  +383.323, E3 -460802.040}
SPL {X  -159.990, Y  +439.778, Z    +0.000, E1  +383.323, E3 -460815.673}
SPL {X  -159.990, Y  +442.945, Z    +0.000, E1  +383.339, E3 -460831.236}
SPL {X  -159.990, Y  +446.037, Z    +0.000, E1  +383.324, E3 -460846.487}
SPL {X  -159.990, Y  +448.341, Z    +0.000, E1  +383.317, E3 -460857.804}
SPL {X  -159.990, Y  +450.345, Z    +0.000, E1  +383.316, E3 -460867.682}
SPL {X  -159.990, Y  +452.828, Z    +0.000, E1  +383.330, E3 -460879.882}
SPL {X  -159.990, Y  +456.338, Z    +0.000, E1  +383.359, E3 -460897.074}
SPL {X  -159.990, Y  +459.480, Z    +0.000, E1  +383.323, E3 -460912.615}
SPL {X  -159.990, Y  +461.803, Z    +0.000, E1  +383.322, E3 -460924.050}
SPL {X  -159.990, Y  +464.971, Z    +0.000, E1  +383.357, E3 -460939.556}
SPL {X  -159.990, Y  +467.934, Z    +0.000, E1  +383.321, E3 -460954.214}
SPL {X  -159.990, Y  +469.939, Z    +0.000, E1  +383.319, E3 -460964.075}
SPL {X  -159.990, Y  +472.144, Z    +0.000, E1  +383.327, E3 -460974.926}
SPL {X  -159.990, Y  +474.152, Z    +0.000, E1  +383.309, E3 -460984.878}
SPL {X  -159.990, Y  +475.762, Z    +0.000, E1  +383.308, E3 -460992.807}
SPL {X  -159.990, Y  +478.041, Z    +0.000, E1  +383.328, E3 -461003.983}
SPL {X  -159.990, Y  +480.905, Z    +0.000, E1  +383.327, E3 -461018.079}
SPL {X  -159.990, Y  +484.251, Z    +0.000, E1  +383.352, E3 -461034.495}
SPL {X  -159.990, Y  +488.031, Z    +0.000, E1  +383.345, E3 -461053.128}
SPL {X  -159.990, Y  +491.121, Z    +0.000, E1  +383.323, E3 -461068.373}
SPL {X  -159.990, Y  +493.610, Z    +0.000, E1  +383.323, E3 -461080.626}
SPL {X  -159.990, Y  +496.863, Z    +0.000, E1  +383.350, E3 -461096.586}
SPL {X  -159.990, Y  +499.995, Z    +0.000, E1  +383.324, E3 -461112.048}
SPL {X  -159.990, Y  +502.341, Z    +0.000, E1  +383.320, E3 -461123.607}
SPL {X  -159.990, Y  +505.377, Z    +0.000, E1  +383.346, E3 -461138.497}
SPL {X  -159.990, Y  +508.024, Z    +0.000, E1  +383.315, E3 -461151.580}
SPL {X  -159.990, Y  +510.344, Z    +0.000, E1  +383.327, E3 -461162.986}
SPL {X  -159.990, Y  +513.289, Z    +0.000, E1  +383.332, E3 -461177.476}
SPL {X  -159.990, Y  +516.195, Z    +0.000, E1  +383.325, E3 -461191.795}
SPL {X  -159.990, Y  +518.925, Z    +0.000, E1  +383.333, E3 -461205.159}
SPL {X  -159.990, Y  +521.408, Z    +0.000, E1  +383.329, E3 -461217.368}
SPL {X  -159.990, Y  +523.942, Z    +0.000, E1  +383.333, E3 -461229.861}
SPL {X  -159.990, Y  +527.007, Z    +0.000, E1  +383.339, E3 -461244.960}
SPL {X  -159.990, Y  +529.993, Z    +0.000, E1  +383.329, E3 -461259.662}
SPL {X  -159.990, Y  +532.441, Z    +0.000, E1  +383.322, E3 -461271.713}
SPL {X  -159.990, Y  +534.618, Z    +0.000, E1  +383.322, E3 -461282.446}
SPL {X  -159.990, Y  +537.024, Z    +0.000, E1  +383.321, E3 -461294.309}
SPL {X  -159.990, Y  +539.129, Z    +0.000, E1  +383.310, E3 -461304.691}
SPL {X  -159.990, Y  +541.183, Z    +0.000, E1  +383.319, E3 -461314.788}
SPL {X  -159.990, Y  +543.647, Z    +0.000, E1  +383.325, E3 -461326.891}
SPL {X  -159.990, Y  +546.832, Z    +0.000, E1  +383.349, E3 -461342.514}
SPL {X  -159.990, Y  +549.756, Z    +0.000, E1  +383.320, E3 -461356.955}
SPL {X  -159.990, Y  +551.655, Z    +0.000, E1  +383.320, E3 -461366.306}
SPL {X  -159.990, Y  +553.711, Z    +0.000, E1  +383.317, E3 -461376.428}
SPL {X  -159.990, Y  +556.481, Z    +0.000, E1  +383.354, E3 -461389.989}
SPL {X  -159.990, Y  +559.475, Z    +0.000, E1  +383.321, E3 -461404.795}
SPL {X  -159.990, Y  +561.830, Z    +0.000, E1  +383.325, E3 -461416.379}
SPL {X  -159.990, Y  +564.273, Z    +0.000, E1  +383.325, E3 -461428.404}
SPL {X  -159.990, Y  +566.342, Z    +0.000, E1  +383.314, E3 -461438.608}
SPL {X  -159.990, Y  +568.184, Z    +0.000, E1  +383.317, E3 -461447.669}
SPL {X  -159.990, Y  +570.314, Z    +0.000, E1  +383.326, E3 -461458.132}
SPL {X  -159.990, Y  +573.444, Z    +0.000, E1  +383.356, E3 -461473.471}
SPL {X  -159.990, Y  +577.161, Z    +0.000, E1  +383.346, E3 -461491.795}
SPL {X  -159.990, Y  +580.840, Z    +0.000, E1  +383.355, E3 -461509.845}
SPL {X  -159.990, Y  +583.973, Z    +0.000, E1  +383.332, E3 -461525.306}
SPL {X  -159.990, Y  +586.020, Z    +0.000, E1  +383.323, E3 -461535.390}
SPL {X  -159.990, Y  +587.711, Z    +0.000, E1  +383.318, E3 -461543.729}
SPL {X  -159.990, Y  +589.763, Z    +0.000, E1  +383.328, E3 -461553.806}
SPL {X  -159.990, Y  +591.698, Z    +0.000, E1  +383.324, E3 -461563.290}
SPL {X  -159.990, Y  +593.847, Z    +0.000, E1  +383.340, E3 -461573.821}
SPL {X  -159.990, Y  +597.018, Z    +0.000, E1  +383.367, E3 -461589.353}
SPL {X  -159.990, Y  +599.887, Z    +0.000, E1  +383.341, E3 -461603.457}
SPL {X  -159.990, Y  +601.949, Z    +0.000, E1  +383.344, E3 -461613.584}
SPL {X  -159.990, Y  +605.106, Z    +0.000, E1  +383.383, E3 -461629.030}
SPL {X  -159.990, Y  +608.111, Z    +0.000, E1  +383.342, E3 -461643.881}
SPL {X  -159.990, Y  +610.073, Z    +0.000, E1  +383.343, E3 -461653.539}
SPL {X  -159.990, Y  +613.021, Z    +0.000, E1  +383.365, E3 -461668.010}
SPL {X  -159.990, Y  +615.657, Z    +0.000, E1  +383.331, E3 -461681.058}
SPL {X  -159.990, Y  +617.658, Z    +0.000, E1  +383.335, E3 -461690.900}
SPL {X  -159.990, Y  +620.788, Z    +0.000, E1  +383.368, E3 -461706.233}
SPL {X  -159.990, Y  +624.347, Z    +0.000, E1  +383.355, E3 -461723.753}
SPL {X  -159.990, Y  +627.144, Z    +0.000, E1  +383.340, E3 -461737.523}
SPL {X  -159.990, Y  +629.284, Z    +0.000, E1  +383.339, E3 -461748.031}
SPL {X  -159.990, Y  +631.206, Z    +0.000, E1  +383.337, E3 -461757.484}
SPL {X  -159.990, Y  +633.318, Z    +0.000, E1  +383.339, E3 -461767.889}
SPL {X  -159.990, Y  +635.650, Z    +0.000, E1  +383.339, E3 -461779.360}
SPL {X  -159.990, Y  +637.597, Z    +0.000, E1  +383.330, E3 -461788.982}
SPL {X  -159.990, Y  +640.369, Z    +0.000, E1  +383.354, E3 -461802.616}
SPL {X  -159.990, Y  +644.241, Z    +0.000, E1  +383.355, E3 -461821.728}
SPL {X  -159.990, Y  +647.550, Z    +0.000, E1  +383.318, E3 -461838.127}
SPL {X  -159.990, Y  +650.790, Z    +0.000, E1  +383.346, E3 -461853.994}
SPL {X  -159.990, Y  +654.543, Z    +0.000, E1  +383.348, E3 -461872.447}
SPL {X  -159.990, Y  +658.319, Z    +0.000, E1  +383.349, E3 -461891.037}
SPL {X  -159.990, Y  +661.392, Z    +0.000, E1  +383.318, E3 -461906.240}
SPL {X  -159.990, Y  +663.662, Z    +0.000, E1  +383.322, E3 -461917.364}
SPL {X  -159.990, Y  +665.964, Z    +0.000, E1  +383.328, E3 -461928.654}
SPL {X  -159.990, Y  +667.870, Z    +0.000, E1  +383.320, E3 -461938.061}
SPL {X  -159.990, Y  +669.861, Z    +0.000, E1  +383.321, E3 -461947.862}
SPL {X  -159.990, Y  +671.893, Z    +0.000, E1  +383.319, E3 -461957.870}
SPL {X  -159.974, Y  +673.789, Z    +0.000, E1  +383.323, E3 -461967.186}
SPL {X  -159.924, Y  +676.110, Z    +0.000, E1  +383.320, E3 -461978.671}
SPL {X  -159.801, Y  +679.265, Z    +0.000, E1  +383.327, E3 -461994.289}
SPL {X  -159.626, Y  +682.287, Z    +0.000, E1  +383.280, E3 -462009.388}
SPL {X  -159.462, Y  +684.486, Z    +0.000, E1  +383.258, E3 -462020.387}
SPL {X  -159.212, Y  +687.262, Z    +0.000, E1  +383.238, E3 -462034.291}
SPL {X  -158.861, Y  +690.475, Z    +0.000, E1  +383.199, E3 -462050.459}
SPL {X  -158.553, Y  +692.896, Z    +0.000, E1  +383.130, E3 -462062.755}
ENDSPLINE

SPLINE
SPL {X  -159.063, Y  +688.696, Z    +0.000, E1  +377.094, E3 -462100.876}
SPL {X  -159.987, Y  +672.488, Z    +0.000, E1  +365.638, E3 -462124.941}
SPL {X  -159.990, Y  +663.928, Z    +0.000, E1  +359.662, E3 -462130.735}
SPL {X  -159.990, Y  +658.009, Z    +0.000, E1  +355.226, E3 -462134.435}
SPL {X  -159.990, Y  +651.879, Z    +0.000, E1  +350.548, E3 -462139.498}
SPL {X  -159.990, Y  +637.832, Z    +0.000, E1  +341.694, E3 -462157.089}
SPL {X  -159.990, Y  +626.634, Z    +0.000, E1  +337.968, E3 -462187.942}
SPL {X  -159.990, Y  +624.622, Z    +0.000, E1  +337.980, E3 -462198.526}
SPL {X  -159.990, Y  +622.489, Z    +0.000, E1  +337.969, E3 -462209.692}
SPL {X  -159.990, Y  +619.267, Z    +0.000, E1  +337.938, E3 -462226.526}
SPL {X  -159.990, Y  +615.467, Z    +0.000, E1  +337.940, E3 -462246.463}
SPL {X  -159.990, Y  +612.600, Z    +0.000, E1  +337.975, E3 -462261.573}
SPL {X  -159.990, Y  +610.646, Z    +0.000, E1  +337.979, E3 -462271.831}
SPL {X  -159.990, Y  +608.810, Z    +0.000, E1  +337.977, E3 -462281.463}
SPL {X  -159.990, Y  +606.481, Z    +0.000, E1  +337.967, E3 -462293.639}
SPL {X  -159.990, Y  +603.419, Z    +0.000, E1  +337.936, E3 -462309.578}
SPL {X  -159.990, Y  +600.642, Z    +0.000, E1  +337.968, E3 -462324.208}
SPL {X  -159.990, Y  +598.568, Z    +0.000, E1  +337.954, E3 -462335.001}
SPL {X  -159.990, Y  +596.440, Z    +0.000, E1  +337.964, E3 -462346.182}
SPL {X  -159.990, Y  +593.768, Z    +0.000, E1  +337.929, E3 -462360.115}
SPL {X  -159.990, Y  +590.068, Z    +0.000, E1  +337.924, E3 -462379.484}
SPL {X  -159.990, Y  +586.620, Z    +0.000, E1  +337.935, E3 -462397.546}
SPL {X  -159.990, Y  +584.080, Z    +0.000, E1  +337.953, E3 -462410.873}
SPL {X  -159.990, Y  +581.924, Z    +0.000, E1  +337.949, E3 -462422.173}
SPL {X  -159.990, Y  +578.886, Z    +0.000, E1  +337.918, E3 -462438.027}
SPL {X  -159.990, Y  +576.252, Z    +0.000, E1  +337.962, E3 -462451.925}
SPL {X  -159.990, Y  +574.188, Z    +0.000, E1  +337.947, E3 -462462.698}
SPL {X  -159.990, Y  +571.954, Z    +0.000, E1  +337.959, E3 -462474.455}
SPL {X  -159.990, Y  +570.110, Z    +0.000, E1  +337.958, E3 -462484.106}
SPL {X  -159.990, Y  +568.165, Z    +0.000, E1  +337.957, E3 -462494.285}
SPL {X  -159.990, Y  +566.106, Z    +0.000, E1  +337.954, E3 -462505.069}
SPL {X  -159.990, Y  +563.259, Z    +0.000, E1  +337.929, E3 -462519.951}
SPL {X  -159.990, Y  +559.661, Z    +0.000, E1  +337.922, E3 -462538.773}
SPL {X  -159.990, Y  +555.965, Z    +0.000, E1  +337.915, E3 -462558.082}
SPL {X  -159.990, Y  +553.115, Z    +0.000, E1  +337.946, E3 -462573.068}
SPL {X  -159.990, Y  +550.886, Z    +0.000, E1  +337.944, E3 -462584.749}
SPL {X  -159.990, Y  +548.568, Z    +0.000, E1  +337.944, E3 -462596.870}
SPL {X  -159.990, Y  +546.537, Z    +0.000, E1  +337.948, E3 -462607.505}
SPL {X  -159.990, Y  +545.062, Z    +0.000, E1  +337.955, E3 -462615.264}
SPL {X  -159.990, Y  +543.060, Z    +0.000, E1  +337.943, E3 -462625.744}
SPL {X  -159.990, Y  +539.928, Z    +0.000, E1  +337.917, E3 -462642.085}
SPL {X  -159.990, Y  +536.935, Z    +0.000, E1  +337.942, E3 -462657.802}
SPL {X  -159.990, Y  +534.656, Z    +0.000, E1  +337.946, E3 -462669.745}
SPL {X  -159.990, Y  +531.679, Z    +0.000, E1  +337.913, E3 -462685.259}
SPL {X  -159.990, Y  +527.941, Z    +0.000, E1  +337.907, E3 -462704.802}
SPL {X  -159.990, Y  +525.053, Z    +0.000, E1  +337.942, E3 -462719.992}
SPL {X  -159.990, Y  +522.838, Z    +0.000, E1  +337.933, E3 -462731.596}
SPL {X  -159.990, Y  +519.698, Z    +0.000, E1  +337.916, E3 -462747.979}
SPL {X  -159.990, Y  +517.251, Z    +0.000, E1  +337.946, E3 -462760.839}
SPL {X  -159.990, Y  +515.568, Z    +0.000, E1  +338.084, E3 -462770.936}
ENDSPLINE

SPLINE
SPL {X  -159.990, Y  +518.374, Z    +0.000, E1  +341.240, E3 -462783.524}
ENDSPLINE

SPLINE
SPL {X  -159.990, Y  +513.606, Z    +0.000, E1  +339.879, E3 -462799.434}
SPL {X  -159.990, Y  +508.660, Z    +0.000, E1  +338.515, E3 -462814.864}
SPL {X  -159.990, Y  +505.237, Z    +0.000, E1  +337.606, E3 -462825.121}
SPL {X  -159.990, Y  +501.963, Z    +0.000, E1  +336.712, E3 -462834.225}
SPL {X  -159.990, Y  +498.406, Z    +0.000, E1  +335.789, E3 -462843.976}
SPL {X  -159.990, Y  +494.693, Z    +0.000, E1  +334.929, E3 -462854.443}
SPL {X  -159.990, Y  +491.649, Z    +0.000, E1  +334.596, E3 -462865.646}
SPL {X  -159.990, Y  +488.807, Z    +0.000, E1  +334.603, E3 -462878.370}
SPL {X  -159.990, Y  +486.070, Z    +0.000, E1  +334.601, E3 -462890.601}
SPL {X  -159.990, Y  +482.821, Z    +0.000, E1  +334.589, E3 -462905.102}
SPL {X  -159.990, Y  +480.183, Z    +0.000, E1  +334.616, E3 -462916.943}
SPL {X  -159.990, Y  +477.508, Z    +0.000, E1  +334.590, E3 -462928.851}
SPL {X  -159.990, Y  +473.634, Z    +0.000, E1  +334.574, E3 -462946.141}
SPL {X  -159.990, Y  +470.047, Z    +0.000, E1  +334.598, E3 -462962.222}
SPL {X  -159.990, Y  +467.082, Z    +0.000, E1  +334.601, E3 -462975.469}
SPL {X  -159.990, Y  +464.063, Z    +0.000, E1  +334.595, E3 -462988.964}
SPL {X  -159.990, Y  +460.712, Z    +0.000, E1  +334.589, E3 -463003.923}
SPL {X  -159.990, Y  +457.497, Z    +0.000, E1  +334.597, E3 -463018.296}
SPL {X  -159.990, Y  +454.323, Z    +0.000, E1  +334.588, E3 -463032.455}
SPL {X  -159.990, Y  +450.823, Z    +0.000, E1  +334.583, E3 -463048.084}
SPL {X  -159.990, Y  +447.982, Z    +0.000, E1  +334.607, E3 -463060.824}
SPL {X  -159.990, Y  +445.108, Z    +0.000, E1  +334.593, E3 -463073.701}
SPL {X  -159.990, Y  +441.797, Z    +0.000, E1  +334.610, E3 -463088.580}
SPL {X  -159.990, Y  +439.442, Z    +0.000, E1  +334.631, E3 -463099.157}
SPL {X  -159.990, Y  +436.316, Z    +0.000, E1  +334.580, E3 -463113.039}
SPL {X  -159.990, Y  +432.613, Z    +0.000, E1  +334.610, E3 -463129.665}
SPL {X  -159.990, Y  +429.827, Z    +0.000, E1  +334.620, E3 -463142.142}
SPL {X  -159.990, Y  +426.865, Z    +0.000, E1  +334.602, E3 -463155.347}
SPL {X  -159.990, Y  +423.417, Z    +0.000, E1  +334.600, E3 -463170.763}
SPL {X  -159.990, Y  +420.283, Z    +0.000, E1  +334.614, E3 -463184.807}
SPL {X  -159.990, Y  +417.103, Z    +0.000, E1  +334.600, E3 -463199.002}
SPL {X  -159.990, Y  +413.684, Z    +0.000, E1  +334.603, E3 -463214.301}
SPL {X  -159.990, Y  +410.645, Z    +0.000, E1  +334.615, E3 -463227.913}
SPL {X  -159.990, Y  +407.450, Z    +0.000, E1  +334.599, E3 -463242.162}
SPL {X  -159.990, Y  +403.513, Z    +0.000, E1  +334.580, E3 -463259.715}
SPL {X  -159.990, Y  +400.403, Z    +0.000, E1  +334.620, E3 -463273.698}
SPL {X  -159.990, Y  +397.743, Z    +0.000, E1  +334.600, E3 -463285.567}
SPL {X  -159.990, Y  +394.848, Z    +0.000, E1  +334.621, E3 -463298.568}
SPL {X  -159.990, Y  +392.473, Z    +0.000, E1  +334.623, E3 -463309.195}
SPL {X  -159.990, Y  +390.187, Z    +0.000, E1  +334.622, E3 -463319.453}
SPL {X  -159.990, Y  +387.503, Z    +0.000, E1  +334.622, E3 -463331.448}
SPL {X  -159.990, Y  +384.711, Z    +0.000, E1  +334.612, E3 -463343.891}
SPL {X  -159.988, Y  +381.794, Z    +0.000, E1  +334.611, E3 -463356.926}
SPL {X  -159.958, Y  +379.279, Z    +0.000, E1  +334.625, E3 -463368.216}
SPL {X  -159.894, Y  +376.959, Z    +0.000, E1  +334.630, E3 -463378.661}
SPL {X  -159.765, Y  +374.027, Z    +0.000, E1  +334.633, E3 -463391.877}
SPL {X  -159.607, Y  +371.442, Z    +0.000, E1  +334.673, E3 -463403.652}
SPL {X  -159.379, Y  +368.534, Z    +0.000, E1  +334.684, E3 -463416.839}
SPL {X  -159.113, Y  +365.767, Z    +0.000, E1  +334.734, E3 -463429.479}
SPL {X  -158.798, Y  +363.007, Z    +0.000, E1  +334.761, E3 -463442.119}
SPL {X  -158.453, Y  +360.380, Z    +0.000, E1  +334.828, E3 -463454.263}
SPL {X  -158.127, Y  +358.155, Z    +0.000, E1  +334.874, E3 -463464.594}
SPL {X  -158.095, Y  +357.947, Z    +0.000, E1  +338.259, E3 -463496.166}
ENDSPLINE

